// TIA Portal V19 export
FUNCTION "AUTO SUBOUTPUT" : Void   // FC15, LAD
{ S7_Optimized_Access := 'TRUE' }
// stored: SetENOAutomatically false
BEGIN

REGION Network 1: SYRUP MFG VESSEL BOTTOM STERROR RUN
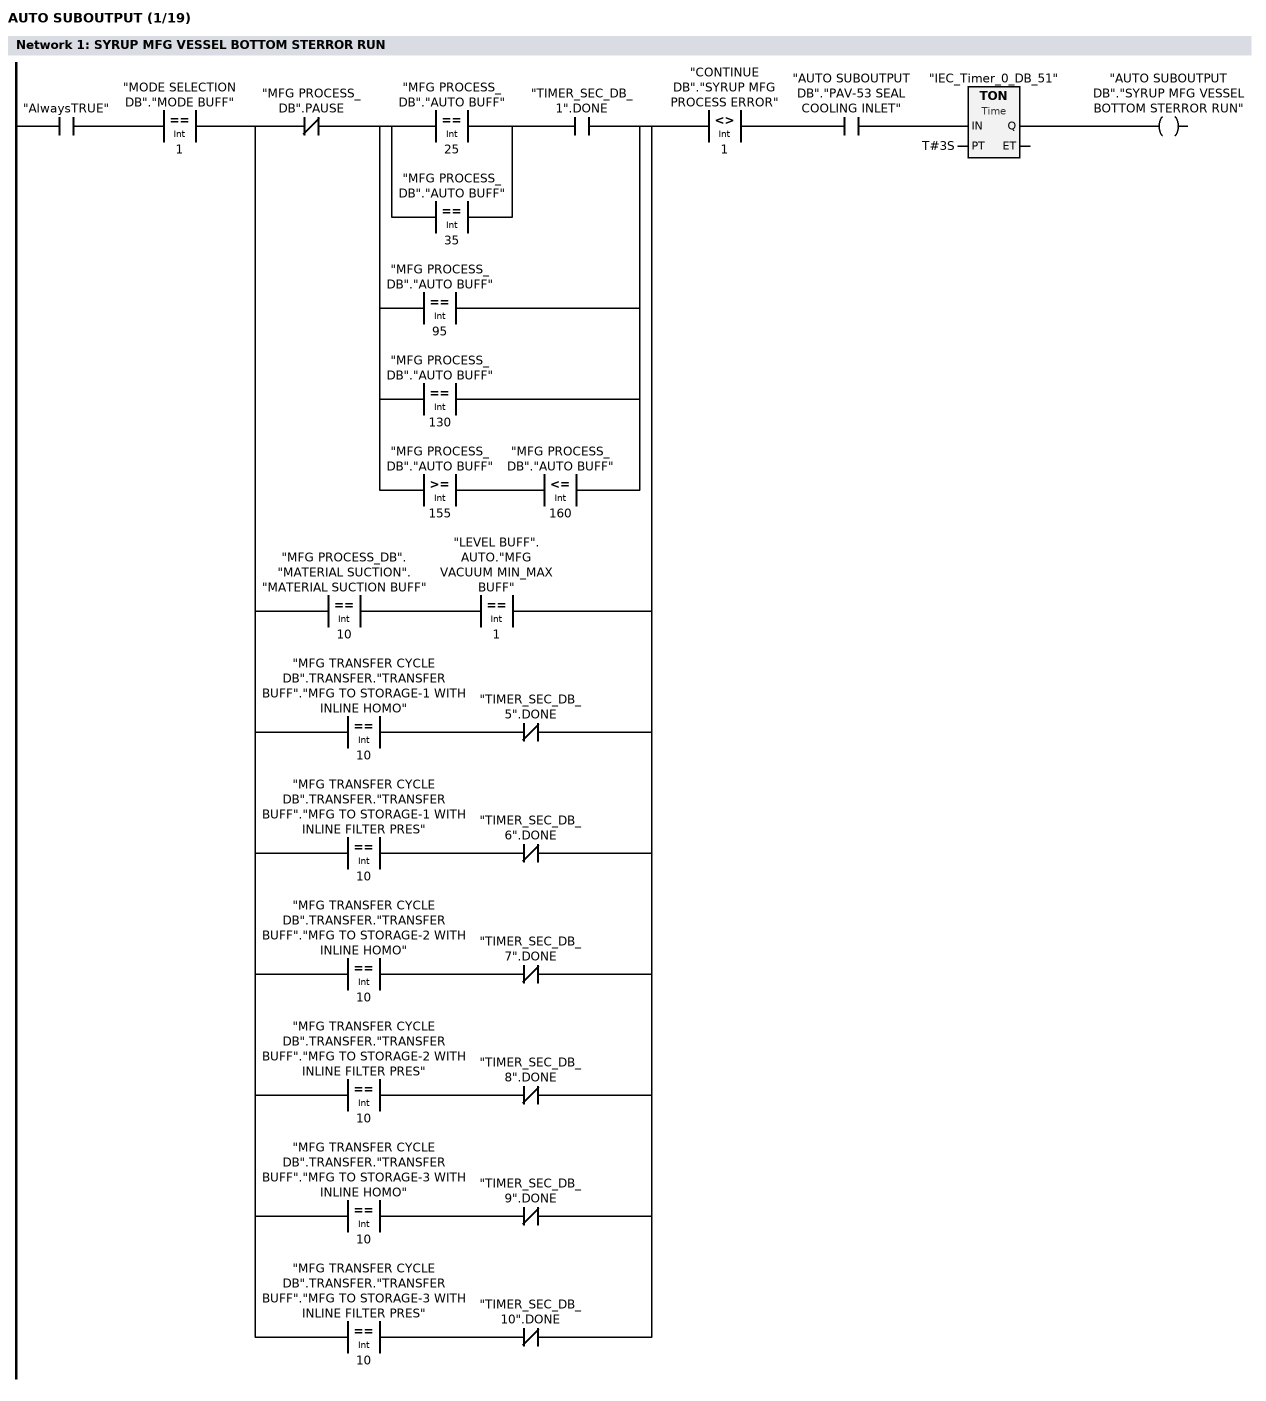
   RUNG wire#powerrail
      Contact( "AlwaysTRUE" )
      { S7_Templates := "SrcType := Int" } EQ_Contact(in1 := "MODE SELECTION DB"."MODE BUFF", in2 := 1)
      wire#w1
      I_Contact( "MFG PROCESS_DB".PAUSE )
      wire#w2
      { S7_Templates := "SrcType := Int" } EQ_Contact(in1 := "MFG PROCESS_DB"."AUTO BUFF", in2 := 25)
      wire#w3
      Contact( "TIMER_SEC_DB_1".DONE )
      wire#w4
      { S7_Templates := "SrcType := Int" } NE_Contact(in1 := "CONTINUE DB"."SYRUP MFG PROCESS ERROR", in2 := 1)
      Contact( "AUTO SUBOUTPUT DB"."PAV-53 SEAL COOLING INLET" )
      { S7_Templates := "time_type := Time" } "IEC_Timer_0_DB_51".TON(pt := T#3S, et =>)
      Coil( "AUTO SUBOUTPUT DB"."SYRUP MFG VESSEL BOTTOM STERROR RUN" )
   END_RUNG
   RUNG wire#w2
      { S7_Templates := "SrcType := Int" } EQ_Contact(in1 := "MFG PROCESS_DB"."AUTO BUFF", in2 := 35)
   END_RUNG wire#w3
   RUNG wire#w2
      { S7_Templates := "SrcType := Int" } EQ_Contact(in1 := "MFG PROCESS_DB"."AUTO BUFF", in2 := 95)
   END_RUNG wire#w4
   RUNG wire#w2
      { S7_Templates := "SrcType := Int" } EQ_Contact(in1 := "MFG PROCESS_DB"."AUTO BUFF", in2 := 130)
   END_RUNG wire#w4
   RUNG wire#w2
      { S7_Templates := "SrcType := Int" } GE_Contact(in1 := "MFG PROCESS_DB"."AUTO BUFF", in2 := 155)
      { S7_Templates := "SrcType := Int" } LE_Contact(in1 := "MFG PROCESS_DB"."AUTO BUFF", in2 := 160)
   END_RUNG wire#w4
   RUNG wire#w1
      { S7_Templates := "SrcType := Int" } EQ_Contact(in1 := "MFG PROCESS_DB"."MATERIAL SUCTION"."MATERIAL SUCTION BUFF", in2 := 10)
      { S7_Templates := "SrcType := Int" } EQ_Contact(in1 := "LEVEL BUFF".AUTO."MFG VACUUM MIN_MAX BUFF", in2 := 1)
   END_RUNG wire#w4
   RUNG wire#w1
      { S7_Templates := "SrcType := Int" } EQ_Contact(in1 := "MFG TRANSFER CYCLE DB".TRANSFER."TRANSFER BUFF"."MFG TO STORAGE-1 WITH INLINE HOMO", in2 := 10)
      I_Contact( "TIMER_SEC_DB_5".DONE )
   END_RUNG wire#w4
   RUNG wire#w1
      { S7_Templates := "SrcType := Int" } EQ_Contact(in1 := "MFG TRANSFER CYCLE DB".TRANSFER."TRANSFER BUFF"."MFG TO STORAGE-1 WITH INLINE FILTER PRES", in2 := 10)
      I_Contact( "TIMER_SEC_DB_6".DONE )
   END_RUNG wire#w4
   RUNG wire#w1
      { S7_Templates := "SrcType := Int" } EQ_Contact(in1 := "MFG TRANSFER CYCLE DB".TRANSFER."TRANSFER BUFF"."MFG TO STORAGE-2 WITH INLINE HOMO", in2 := 10)
      I_Contact( "TIMER_SEC_DB_7".DONE )
   END_RUNG wire#w4
   RUNG wire#w1
      { S7_Templates := "SrcType := Int" } EQ_Contact(in1 := "MFG TRANSFER CYCLE DB".TRANSFER."TRANSFER BUFF"."MFG TO STORAGE-2 WITH INLINE FILTER PRES", in2 := 10)
      I_Contact( "TIMER_SEC_DB_8".DONE )
   END_RUNG wire#w4
   RUNG wire#w1
      { S7_Templates := "SrcType := Int" } EQ_Contact(in1 := "MFG TRANSFER CYCLE DB".TRANSFER."TRANSFER BUFF"."MFG TO STORAGE-3 WITH INLINE HOMO", in2 := 10)
      I_Contact( "TIMER_SEC_DB_9".DONE )
   END_RUNG wire#w4
   RUNG wire#w1
      { S7_Templates := "SrcType := Int" } EQ_Contact(in1 := "MFG TRANSFER CYCLE DB".TRANSFER."TRANSFER BUFF"."MFG TO STORAGE-3 WITH INLINE FILTER PRES", in2 := 10)
      I_Contact( "TIMER_SEC_DB_10".DONE )
   END_RUNG wire#w4
   // the same network as SCL:
   "IEC_Timer_0_DB_51".TON(IN := "AlwaysTRUE" AND ("MODE SELECTION DB"."MODE BUFF" = 1) AND ((NOT "MFG PROCESS_DB".PAUSE AND (((("MFG PROCESS_DB"."AUTO BUFF" = 25) OR ("MFG PROCESS_DB"."AUTO BUFF" = 35)) AND "TIMER_SEC_DB_1".DONE) OR ("MFG PROCESS_DB"."AUTO BUFF" = 95) OR ("MFG PROCESS_DB"."AUTO BUFF" = 130) OR (("MFG PROCESS_DB"."AUTO BUFF" >= 155) AND ("MFG PROCESS_DB"."AUTO BUFF" <= 160)))) OR (("MFG PROCESS_DB"."MATERIAL SUCTION"."MATERIAL SUCTION BUFF" = 10) AND ("LEVEL BUFF".AUTO."MFG VACUUM MIN_MAX BUFF" = 1)) OR (("MFG TRANSFER CYCLE DB".TRANSFER."TRANSFER BUFF"."MFG TO STORAGE-1 WITH INLINE HOMO" = 10) AND NOT "TIMER_SEC_DB_5".DONE) OR (("MFG TRANSFER CYCLE DB".TRANSFER."TRANSFER BUFF"."MFG TO STORAGE-1 WITH INLINE FILTER PRES" = 10) AND NOT "TIMER_SEC_DB_6".DONE) OR (("MFG TRANSFER CYCLE DB".TRANSFER."TRANSFER BUFF"."MFG TO STORAGE-2 WITH INLINE HOMO" = 10) AND NOT "TIMER_SEC_DB_7".DONE) OR (("MFG TRANSFER CYCLE DB".TRANSFER."TRANSFER BUFF"."MFG TO STORAGE-2 WITH INLINE FILTER PRES" = 10) AND NOT "TIMER_SEC_DB_8".DONE) OR (("MFG TRANSFER CYCLE DB".TRANSFER."TRANSFER BUFF"."MFG TO STORAGE-3 WITH INLINE HOMO" = 10) AND NOT "TIMER_SEC_DB_9".DONE) OR (("MFG TRANSFER CYCLE DB".TRANSFER."TRANSFER BUFF"."MFG TO STORAGE-3 WITH INLINE FILTER PRES" = 10) AND NOT "TIMER_SEC_DB_10".DONE)) AND ("CONTINUE DB"."SYRUP MFG PROCESS ERROR" <> 1) AND "AUTO SUBOUTPUT DB"."PAV-53 SEAL COOLING INLET",
                           PT := T#3S);
   "AUTO SUBOUTPUT DB"."SYRUP MFG VESSEL BOTTOM STERROR RUN" := "IEC_Timer_0_DB_51".Q;
END_REGION

REGION Network 2: PREMIXING VESSEL BOTTOM STERROR RUN
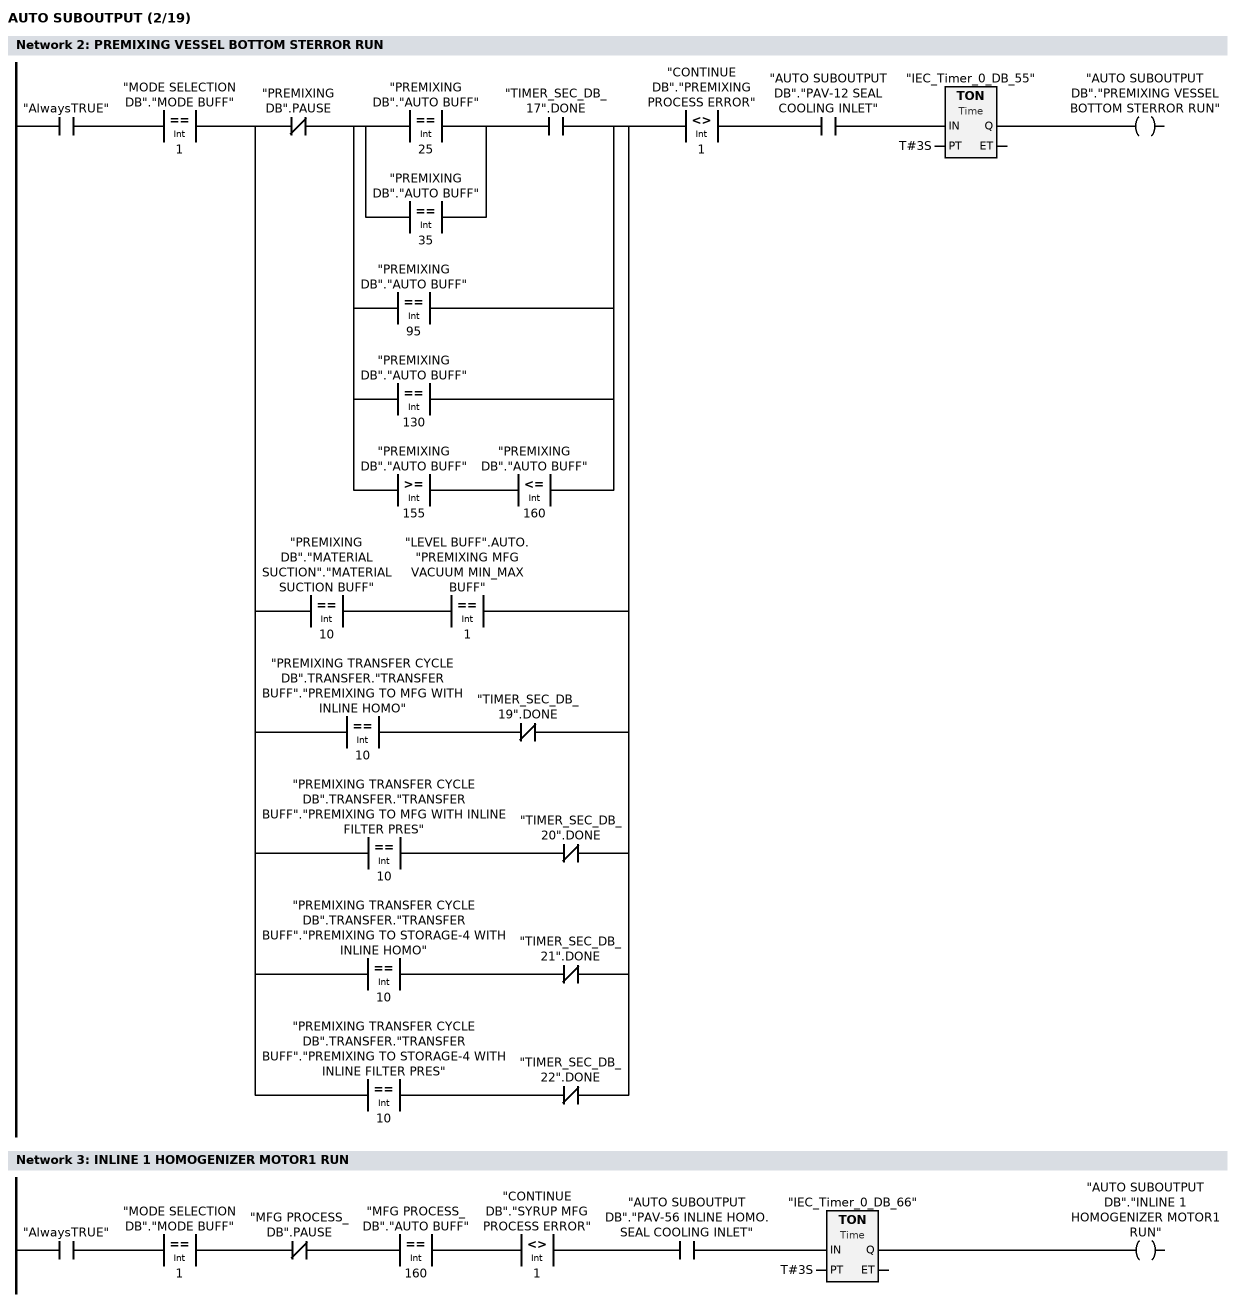
   RUNG wire#powerrail
      Contact( "AlwaysTRUE" )
      { S7_Templates := "SrcType := Int" } EQ_Contact(in1 := "MODE SELECTION DB"."MODE BUFF", in2 := 1)
      wire#w1
      I_Contact( "PREMIXING DB".PAUSE )
      wire#w2
      { S7_Templates := "SrcType := Int" } EQ_Contact(in1 := "PREMIXING DB"."AUTO BUFF", in2 := 25)
      wire#w3
      Contact( "TIMER_SEC_DB_17".DONE )
      wire#w4
      { S7_Templates := "SrcType := Int" } NE_Contact(in1 := "CONTINUE DB"."PREMIXING PROCESS ERROR", in2 := 1)
      Contact( "AUTO SUBOUTPUT DB"."PAV-12 SEAL COOLING INLET" )
      { S7_Templates := "time_type := Time" } "IEC_Timer_0_DB_55".TON(pt := T#3S, et =>)
      Coil( "AUTO SUBOUTPUT DB"."PREMIXING VESSEL BOTTOM STERROR RUN" )
   END_RUNG
   RUNG wire#w2
      { S7_Templates := "SrcType := Int" } EQ_Contact(in1 := "PREMIXING DB"."AUTO BUFF", in2 := 35)
   END_RUNG wire#w3
   RUNG wire#w2
      { S7_Templates := "SrcType := Int" } EQ_Contact(in1 := "PREMIXING DB"."AUTO BUFF", in2 := 95)
   END_RUNG wire#w4
   RUNG wire#w2
      { S7_Templates := "SrcType := Int" } EQ_Contact(in1 := "PREMIXING DB"."AUTO BUFF", in2 := 130)
   END_RUNG wire#w4
   RUNG wire#w2
      { S7_Templates := "SrcType := Int" } GE_Contact(in1 := "PREMIXING DB"."AUTO BUFF", in2 := 155)
      { S7_Templates := "SrcType := Int" } LE_Contact(in1 := "PREMIXING DB"."AUTO BUFF", in2 := 160)
   END_RUNG wire#w4
   RUNG wire#w1
      { S7_Templates := "SrcType := Int" } EQ_Contact(in1 := "PREMIXING DB"."MATERIAL SUCTION"."MATERIAL SUCTION BUFF", in2 := 10)
      { S7_Templates := "SrcType := Int" } EQ_Contact(in1 := "LEVEL BUFF".AUTO."PREMIXING MFG VACUUM MIN_MAX BUFF", in2 := 1)
   END_RUNG wire#w4
   RUNG wire#w1
      { S7_Templates := "SrcType := Int" } EQ_Contact(in1 := "PREMIXING TRANSFER CYCLE DB".TRANSFER."TRANSFER BUFF"."PREMIXING TO MFG WITH INLINE HOMO", in2 := 10)
      I_Contact( "TIMER_SEC_DB_19".DONE )
   END_RUNG wire#w4
   RUNG wire#w1
      { S7_Templates := "SrcType := Int" } EQ_Contact(in1 := "PREMIXING TRANSFER CYCLE DB".TRANSFER."TRANSFER BUFF"."PREMIXING TO MFG WITH INLINE FILTER PRES", in2 := 10)
      I_Contact( "TIMER_SEC_DB_20".DONE )
   END_RUNG wire#w4
   RUNG wire#w1
      { S7_Templates := "SrcType := Int" } EQ_Contact(in1 := "PREMIXING TRANSFER CYCLE DB".TRANSFER."TRANSFER BUFF"."PREMIXING TO STORAGE-4 WITH INLINE HOMO", in2 := 10)
      I_Contact( "TIMER_SEC_DB_21".DONE )
   END_RUNG wire#w4
   RUNG wire#w1
      { S7_Templates := "SrcType := Int" } EQ_Contact(in1 := "PREMIXING TRANSFER CYCLE DB".TRANSFER."TRANSFER BUFF"."PREMIXING TO STORAGE-4 WITH INLINE FILTER PRES", in2 := 10)
      I_Contact( "TIMER_SEC_DB_22".DONE )
   END_RUNG wire#w4
   // the same network as SCL:
   "IEC_Timer_0_DB_55".TON(IN := "AlwaysTRUE" AND ("MODE SELECTION DB"."MODE BUFF" = 1) AND ((NOT "PREMIXING DB".PAUSE AND (((("PREMIXING DB"."AUTO BUFF" = 25) OR ("PREMIXING DB"."AUTO BUFF" = 35)) AND "TIMER_SEC_DB_17".DONE) OR ("PREMIXING DB"."AUTO BUFF" = 95) OR ("PREMIXING DB"."AUTO BUFF" = 130) OR (("PREMIXING DB"."AUTO BUFF" >= 155) AND ("PREMIXING DB"."AUTO BUFF" <= 160)))) OR (("PREMIXING DB"."MATERIAL SUCTION"."MATERIAL SUCTION BUFF" = 10) AND ("LEVEL BUFF".AUTO."PREMIXING MFG VACUUM MIN_MAX BUFF" = 1)) OR (("PREMIXING TRANSFER CYCLE DB".TRANSFER."TRANSFER BUFF"."PREMIXING TO MFG WITH INLINE HOMO" = 10) AND NOT "TIMER_SEC_DB_19".DONE) OR (("PREMIXING TRANSFER CYCLE DB".TRANSFER."TRANSFER BUFF"."PREMIXING TO MFG WITH INLINE FILTER PRES" = 10) AND NOT "TIMER_SEC_DB_20".DONE) OR (("PREMIXING TRANSFER CYCLE DB".TRANSFER."TRANSFER BUFF"."PREMIXING TO STORAGE-4 WITH INLINE HOMO" = 10) AND NOT "TIMER_SEC_DB_21".DONE) OR (("PREMIXING TRANSFER CYCLE DB".TRANSFER."TRANSFER BUFF"."PREMIXING TO STORAGE-4 WITH INLINE FILTER PRES" = 10) AND NOT "TIMER_SEC_DB_22".DONE)) AND ("CONTINUE DB"."PREMIXING PROCESS ERROR" <> 1) AND "AUTO SUBOUTPUT DB"."PAV-12 SEAL COOLING INLET",
                           PT := T#3S);
   "AUTO SUBOUTPUT DB"."PREMIXING VESSEL BOTTOM STERROR RUN" := "IEC_Timer_0_DB_55".Q;
END_REGION

REGION Network 3: INLINE 1 HOMOGENIZER MOTOR1 RUN
   RUNG wire#powerrail
      Contact( "AlwaysTRUE" )
      { S7_Templates := "SrcType := Int" } EQ_Contact(in1 := "MODE SELECTION DB"."MODE BUFF", in2 := 1)
      I_Contact( "MFG PROCESS_DB".PAUSE )
      { S7_Templates := "SrcType := Int" } EQ_Contact(in1 := "MFG PROCESS_DB"."AUTO BUFF", in2 := 160)
      { S7_Templates := "SrcType := Int" } NE_Contact(in1 := "CONTINUE DB"."SYRUP MFG PROCESS ERROR", in2 := 1)
      Contact( "AUTO SUBOUTPUT DB"."PAV-56 INLINE HOMO. SEAL COOLING INLET" )
      { S7_Templates := "time_type := Time" } "IEC_Timer_0_DB_66".TON(pt := T#3S, et =>)
      Coil( "AUTO SUBOUTPUT DB"."INLINE 1 HOMOGENIZER MOTOR1 RUN" )
   END_RUNG
   // the same network as SCL:
   "IEC_Timer_0_DB_66".TON(IN := "AlwaysTRUE" AND ("MODE SELECTION DB"."MODE BUFF" = 1) AND NOT "MFG PROCESS_DB".PAUSE AND ("MFG PROCESS_DB"."AUTO BUFF" = 160) AND ("CONTINUE DB"."SYRUP MFG PROCESS ERROR" <> 1) AND "AUTO SUBOUTPUT DB"."PAV-56 INLINE HOMO. SEAL COOLING INLET",
                           PT := T#3S);
   "AUTO SUBOUTPUT DB"."INLINE 1 HOMOGENIZER MOTOR1 RUN" := "IEC_Timer_0_DB_66".Q;
END_REGION

REGION Network 4: INLINE 2 HOMOGENIZER MOTOR 2 RUN
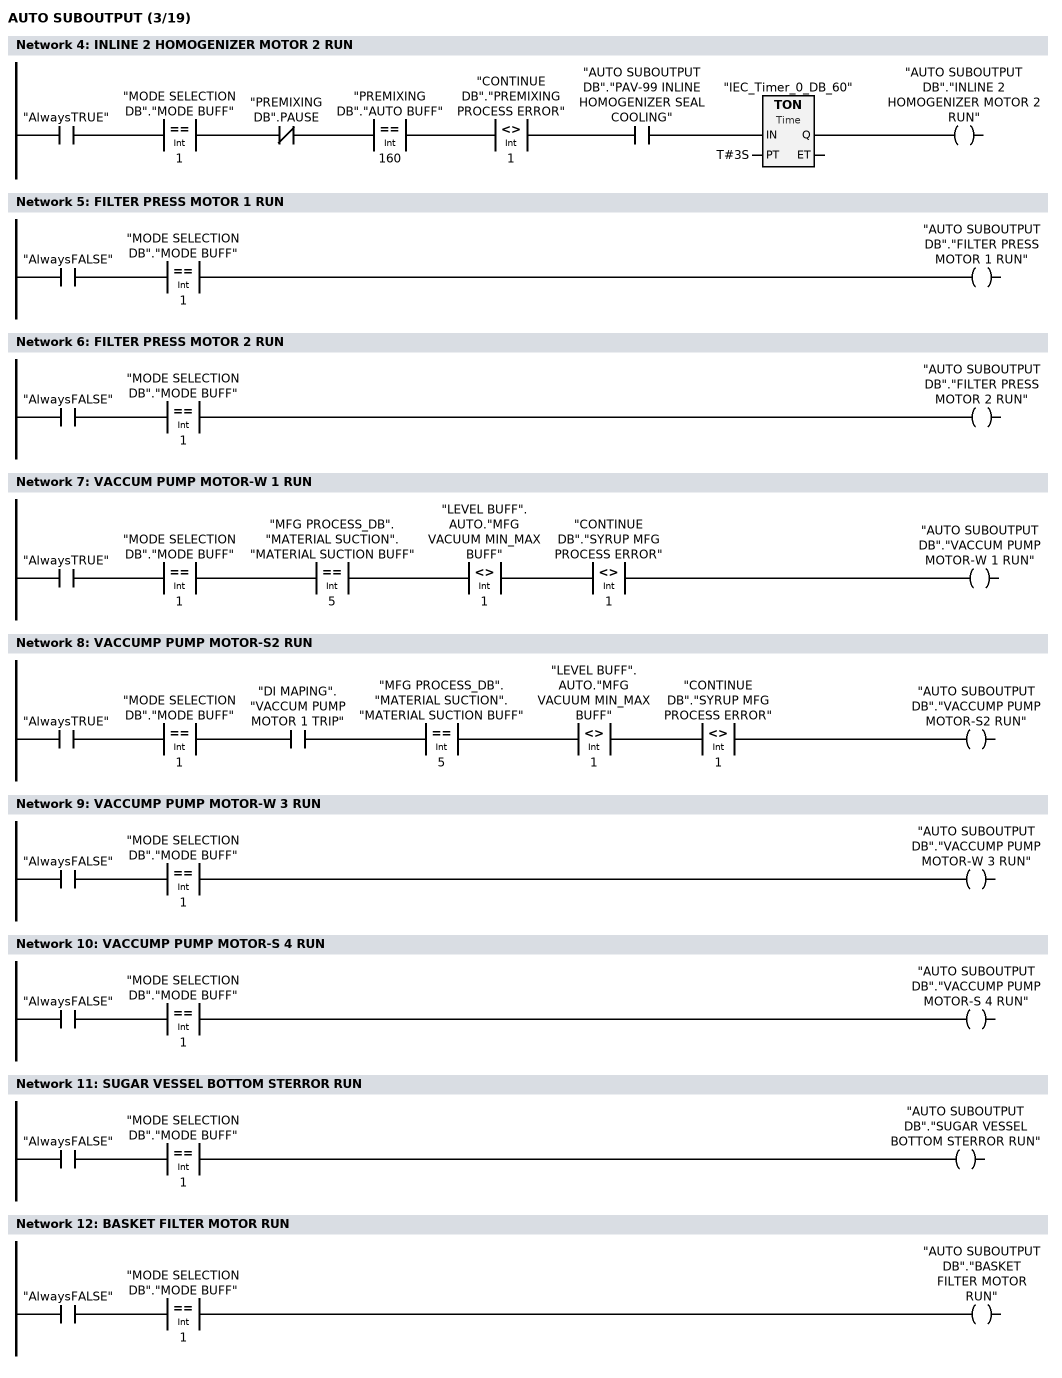
   RUNG wire#powerrail
      Contact( "AlwaysTRUE" )
      { S7_Templates := "SrcType := Int" } EQ_Contact(in1 := "MODE SELECTION DB"."MODE BUFF", in2 := 1)
      I_Contact( "PREMIXING DB".PAUSE )
      { S7_Templates := "SrcType := Int" } EQ_Contact(in1 := "PREMIXING DB"."AUTO BUFF", in2 := 160)
      { S7_Templates := "SrcType := Int" } NE_Contact(in1 := "CONTINUE DB"."PREMIXING PROCESS ERROR", in2 := 1)
      Contact( "AUTO SUBOUTPUT DB"."PAV-99 INLINE HOMOGENIZER SEAL COOLING" )
      { S7_Templates := "time_type := Time" } "IEC_Timer_0_DB_60".TON(pt := T#3S, et =>)
      Coil( "AUTO SUBOUTPUT DB"."INLINE 2 HOMOGENIZER MOTOR 2 RUN" )
   END_RUNG
   // the same network as SCL:
   "IEC_Timer_0_DB_60".TON(IN := "AlwaysTRUE" AND ("MODE SELECTION DB"."MODE BUFF" = 1) AND NOT "PREMIXING DB".PAUSE AND ("PREMIXING DB"."AUTO BUFF" = 160) AND ("CONTINUE DB"."PREMIXING PROCESS ERROR" <> 1) AND "AUTO SUBOUTPUT DB"."PAV-99 INLINE HOMOGENIZER SEAL COOLING",
                           PT := T#3S);
   "AUTO SUBOUTPUT DB"."INLINE 2 HOMOGENIZER MOTOR 2 RUN" := "IEC_Timer_0_DB_60".Q;
END_REGION

REGION Network 5: FILTER PRESS MOTOR 1 RUN
   RUNG wire#powerrail
      Contact( "AlwaysFALSE" )
      { S7_Templates := "SrcType := Int" } EQ_Contact(in1 := "MODE SELECTION DB"."MODE BUFF", in2 := 1)
      Coil( "AUTO SUBOUTPUT DB"."FILTER PRESS MOTOR 1 RUN" )
   END_RUNG
   // the same network as SCL:
   "AUTO SUBOUTPUT DB"."FILTER PRESS MOTOR 1 RUN" := "AlwaysFALSE" AND ("MODE SELECTION DB"."MODE BUFF" = 1);
END_REGION

REGION Network 6: FILTER PRESS MOTOR 2 RUN
   RUNG wire#powerrail
      Contact( "AlwaysFALSE" )
      { S7_Templates := "SrcType := Int" } EQ_Contact(in1 := "MODE SELECTION DB"."MODE BUFF", in2 := 1)
      Coil( "AUTO SUBOUTPUT DB"."FILTER PRESS MOTOR 2 RUN" )
   END_RUNG
   // the same network as SCL:
   "AUTO SUBOUTPUT DB"."FILTER PRESS MOTOR 2 RUN" := "AlwaysFALSE" AND ("MODE SELECTION DB"."MODE BUFF" = 1);
END_REGION

REGION Network 7: VACCUM PUMP MOTOR-W 1 RUN
   RUNG wire#powerrail
      Contact( "AlwaysTRUE" )
      { S7_Templates := "SrcType := Int" } EQ_Contact(in1 := "MODE SELECTION DB"."MODE BUFF", in2 := 1)
      { S7_Templates := "SrcType := Int" } EQ_Contact(in1 := "MFG PROCESS_DB"."MATERIAL SUCTION"."MATERIAL SUCTION BUFF", in2 := 5)
      { S7_Templates := "SrcType := Int" } NE_Contact(in1 := "LEVEL BUFF".AUTO."MFG VACUUM MIN_MAX BUFF", in2 := 1)
      { S7_Templates := "SrcType := Int" } NE_Contact(in1 := "CONTINUE DB"."SYRUP MFG PROCESS ERROR", in2 := 1)
      Coil( "AUTO SUBOUTPUT DB"."VACCUM PUMP MOTOR-W 1 RUN" )
   END_RUNG
   // the same network as SCL:
   "AUTO SUBOUTPUT DB"."VACCUM PUMP MOTOR-W 1 RUN" := "AlwaysTRUE" AND ("MODE SELECTION DB"."MODE BUFF" = 1) AND ("MFG PROCESS_DB"."MATERIAL SUCTION"."MATERIAL SUCTION BUFF" = 5) AND ("LEVEL BUFF".AUTO."MFG VACUUM MIN_MAX BUFF" <> 1) AND ("CONTINUE DB"."SYRUP MFG PROCESS ERROR" <> 1);
END_REGION

REGION Network 8: VACCUMP PUMP MOTOR-S2 RUN
   RUNG wire#powerrail
      Contact( "AlwaysTRUE" )
      { S7_Templates := "SrcType := Int" } EQ_Contact(in1 := "MODE SELECTION DB"."MODE BUFF", in2 := 1)
      Contact( "DI MAPING"."VACCUM PUMP MOTOR 1 TRIP" )
      { S7_Templates := "SrcType := Int" } EQ_Contact(in1 := "MFG PROCESS_DB"."MATERIAL SUCTION"."MATERIAL SUCTION BUFF", in2 := 5)
      { S7_Templates := "SrcType := Int" } NE_Contact(in1 := "LEVEL BUFF".AUTO."MFG VACUUM MIN_MAX BUFF", in2 := 1)
      { S7_Templates := "SrcType := Int" } NE_Contact(in1 := "CONTINUE DB"."SYRUP MFG PROCESS ERROR", in2 := 1)
      Coil( "AUTO SUBOUTPUT DB"."VACCUMP PUMP MOTOR-S2 RUN" )
   END_RUNG
   // the same network as SCL:
   "AUTO SUBOUTPUT DB"."VACCUMP PUMP MOTOR-S2 RUN" := "AlwaysTRUE" AND ("MODE SELECTION DB"."MODE BUFF" = 1) AND "DI MAPING"."VACCUM PUMP MOTOR 1 TRIP" AND ("MFG PROCESS_DB"."MATERIAL SUCTION"."MATERIAL SUCTION BUFF" = 5) AND ("LEVEL BUFF".AUTO."MFG VACUUM MIN_MAX BUFF" <> 1) AND ("CONTINUE DB"."SYRUP MFG PROCESS ERROR" <> 1);
END_REGION

REGION Network 9: VACCUMP PUMP MOTOR-W 3 RUN
   RUNG wire#powerrail
      Contact( "AlwaysFALSE" )
      { S7_Templates := "SrcType := Int" } EQ_Contact(in1 := "MODE SELECTION DB"."MODE BUFF", in2 := 1)
      Coil( "AUTO SUBOUTPUT DB"."VACCUMP PUMP MOTOR-W 3 RUN" )
   END_RUNG
   // the same network as SCL:
   "AUTO SUBOUTPUT DB"."VACCUMP PUMP MOTOR-W 3 RUN" := "AlwaysFALSE" AND ("MODE SELECTION DB"."MODE BUFF" = 1);
END_REGION

REGION Network 10: VACCUMP PUMP MOTOR-S 4 RUN
   RUNG wire#powerrail
      Contact( "AlwaysFALSE" )
      { S7_Templates := "SrcType := Int" } EQ_Contact(in1 := "MODE SELECTION DB"."MODE BUFF", in2 := 1)
      Coil( "AUTO SUBOUTPUT DB"."VACCUMP PUMP MOTOR-S 4 RUN" )
   END_RUNG
   // the same network as SCL:
   "AUTO SUBOUTPUT DB"."VACCUMP PUMP MOTOR-S 4 RUN" := "AlwaysFALSE" AND ("MODE SELECTION DB"."MODE BUFF" = 1);
END_REGION

REGION Network 11: SUGAR VESSEL BOTTOM STERROR RUN
   RUNG wire#powerrail
      Contact( "AlwaysFALSE" )
      { S7_Templates := "SrcType := Int" } EQ_Contact(in1 := "MODE SELECTION DB"."MODE BUFF", in2 := 1)
      Coil( "AUTO SUBOUTPUT DB"."SUGAR VESSEL BOTTOM STERROR RUN" )
   END_RUNG
   // the same network as SCL:
   "AUTO SUBOUTPUT DB"."SUGAR VESSEL BOTTOM STERROR RUN" := "AlwaysFALSE" AND ("MODE SELECTION DB"."MODE BUFF" = 1);
END_REGION

REGION Network 12: BASKET FILTER MOTOR RUN
   RUNG wire#powerrail
      Contact( "AlwaysFALSE" )
      { S7_Templates := "SrcType := Int" } EQ_Contact(in1 := "MODE SELECTION DB"."MODE BUFF", in2 := 1)
      Coil( "AUTO SUBOUTPUT DB"."BASKET FILTER MOTOR RUN" )
   END_RUNG
   // the same network as SCL:
   "AUTO SUBOUTPUT DB"."BASKET FILTER MOTOR RUN" := "AlwaysFALSE" AND ("MODE SELECTION DB"."MODE BUFF" = 1);
END_REGION

REGION Network 13: PBV-01 INGREDIENT INLET
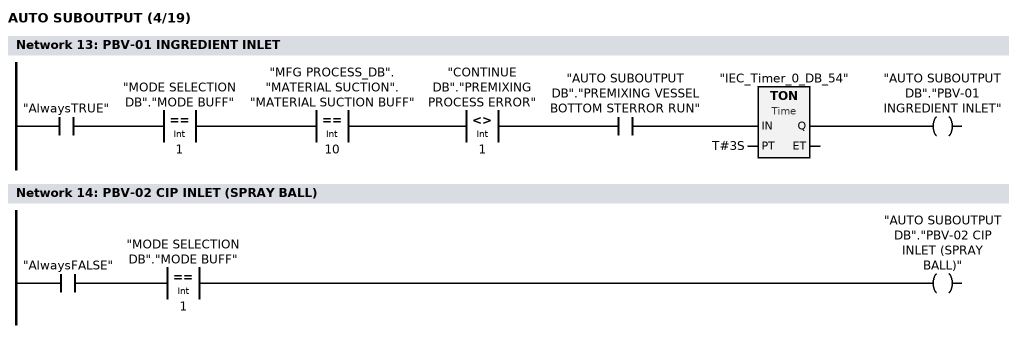
   RUNG wire#powerrail
      Contact( "AlwaysTRUE" )
      { S7_Templates := "SrcType := Int" } EQ_Contact(in1 := "MODE SELECTION DB"."MODE BUFF", in2 := 1)
      { S7_Templates := "SrcType := Int" } EQ_Contact(in1 := "MFG PROCESS_DB"."MATERIAL SUCTION"."MATERIAL SUCTION BUFF", in2 := 10)
      { S7_Templates := "SrcType := Int" } NE_Contact(in1 := "CONTINUE DB"."PREMIXING PROCESS ERROR", in2 := 1)
      Contact( "AUTO SUBOUTPUT DB"."PREMIXING VESSEL BOTTOM STERROR RUN" )
      { S7_Templates := "time_type := Time" } "IEC_Timer_0_DB_54".TON(pt := T#3S, et =>)
      Coil( "AUTO SUBOUTPUT DB"."PBV-01 INGREDIENT INLET" )
   END_RUNG
   // the same network as SCL:
   "IEC_Timer_0_DB_54".TON(IN := "AlwaysTRUE" AND ("MODE SELECTION DB"."MODE BUFF" = 1) AND ("MFG PROCESS_DB"."MATERIAL SUCTION"."MATERIAL SUCTION BUFF" = 10) AND ("CONTINUE DB"."PREMIXING PROCESS ERROR" <> 1) AND "AUTO SUBOUTPUT DB"."PREMIXING VESSEL BOTTOM STERROR RUN",
                           PT := T#3S);
   "AUTO SUBOUTPUT DB"."PBV-01 INGREDIENT INLET" := "IEC_Timer_0_DB_54".Q;
END_REGION

REGION Network 14: PBV-02 CIP INLET (SPRAY BALL)
   RUNG wire#powerrail
      Contact( "AlwaysFALSE" )
      { S7_Templates := "SrcType := Int" } EQ_Contact(in1 := "MODE SELECTION DB"."MODE BUFF", in2 := 1)
      Coil( "AUTO SUBOUTPUT DB"."PBV-02 CIP INLET (SPRAY BALL)" )
   END_RUNG
   // the same network as SCL:
   "AUTO SUBOUTPUT DB"."PBV-02 CIP INLET (SPRAY BALL)" := "AlwaysFALSE" AND ("MODE SELECTION DB"."MODE BUFF" = 1);
END_REGION

REGION Network 15: PBV-03 VENT FILTER ISOLATION
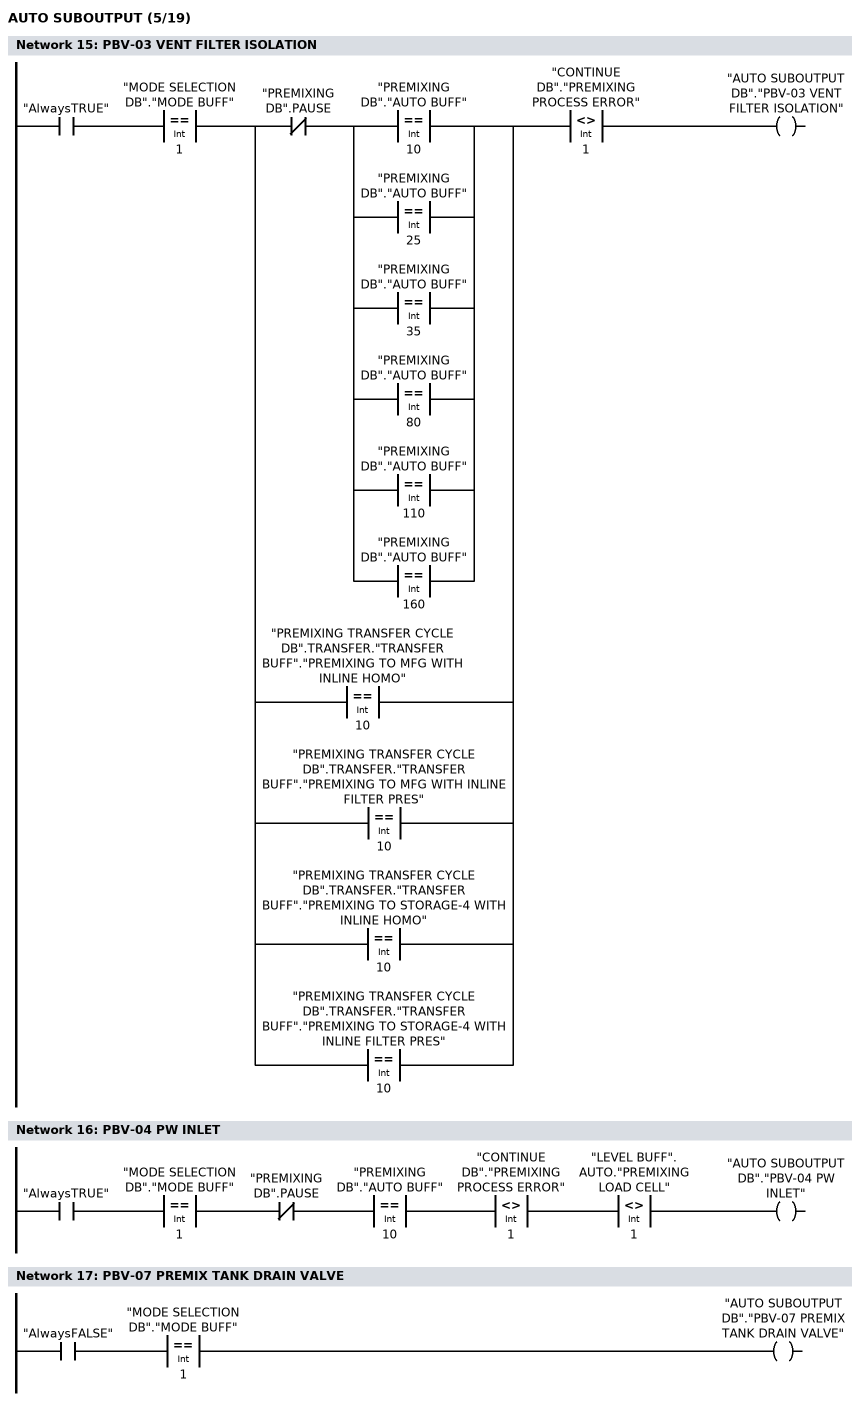
   RUNG wire#powerrail
      Contact( "AlwaysTRUE" )
      { S7_Templates := "SrcType := Int" } EQ_Contact(in1 := "MODE SELECTION DB"."MODE BUFF", in2 := 1)
      wire#w1
      I_Contact( "PREMIXING DB".PAUSE )
      wire#w2
      { S7_Templates := "SrcType := Int" } EQ_Contact(in1 := "PREMIXING DB"."AUTO BUFF", in2 := 10)
      wire#w3
      { S7_Templates := "SrcType := Int" } NE_Contact(in1 := "CONTINUE DB"."PREMIXING PROCESS ERROR", in2 := 1)
      Coil( "AUTO SUBOUTPUT DB"."PBV-03 VENT FILTER ISOLATION" )
   END_RUNG
   RUNG wire#w2
      { S7_Templates := "SrcType := Int" } EQ_Contact(in1 := "PREMIXING DB"."AUTO BUFF", in2 := 25)
   END_RUNG wire#w3
   RUNG wire#w2
      { S7_Templates := "SrcType := Int" } EQ_Contact(in1 := "PREMIXING DB"."AUTO BUFF", in2 := 35)
   END_RUNG wire#w3
   RUNG wire#w2
      { S7_Templates := "SrcType := Int" } EQ_Contact(in1 := "PREMIXING DB"."AUTO BUFF", in2 := 80)
   END_RUNG wire#w3
   RUNG wire#w2
      { S7_Templates := "SrcType := Int" } EQ_Contact(in1 := "PREMIXING DB"."AUTO BUFF", in2 := 110)
   END_RUNG wire#w3
   RUNG wire#w2
      { S7_Templates := "SrcType := Int" } EQ_Contact(in1 := "PREMIXING DB"."AUTO BUFF", in2 := 160)
   END_RUNG wire#w3
   RUNG wire#w1
      { S7_Templates := "SrcType := Int" } EQ_Contact(in1 := "PREMIXING TRANSFER CYCLE DB".TRANSFER."TRANSFER BUFF"."PREMIXING TO MFG WITH INLINE HOMO", in2 := 10)
   END_RUNG wire#w3
   RUNG wire#w1
      { S7_Templates := "SrcType := Int" } EQ_Contact(in1 := "PREMIXING TRANSFER CYCLE DB".TRANSFER."TRANSFER BUFF"."PREMIXING TO MFG WITH INLINE FILTER PRES", in2 := 10)
   END_RUNG wire#w3
   RUNG wire#w1
      { S7_Templates := "SrcType := Int" } EQ_Contact(in1 := "PREMIXING TRANSFER CYCLE DB".TRANSFER."TRANSFER BUFF"."PREMIXING TO STORAGE-4 WITH INLINE HOMO", in2 := 10)
   END_RUNG wire#w3
   RUNG wire#w1
      { S7_Templates := "SrcType := Int" } EQ_Contact(in1 := "PREMIXING TRANSFER CYCLE DB".TRANSFER."TRANSFER BUFF"."PREMIXING TO STORAGE-4 WITH INLINE FILTER PRES", in2 := 10)
   END_RUNG wire#w3
   // the same network as SCL:
   "AUTO SUBOUTPUT DB"."PBV-03 VENT FILTER ISOLATION" := "AlwaysTRUE" AND ("MODE SELECTION DB"."MODE BUFF" = 1) AND ((NOT "PREMIXING DB".PAUSE AND (("PREMIXING DB"."AUTO BUFF" = 10) OR ("PREMIXING DB"."AUTO BUFF" = 25) OR ("PREMIXING DB"."AUTO BUFF" = 35) OR ("PREMIXING DB"."AUTO BUFF" = 80) OR ("PREMIXING DB"."AUTO BUFF" = 110) OR ("PREMIXING DB"."AUTO BUFF" = 160))) OR ("PREMIXING TRANSFER CYCLE DB".TRANSFER."TRANSFER BUFF"."PREMIXING TO MFG WITH INLINE HOMO" = 10) OR ("PREMIXING TRANSFER CYCLE DB".TRANSFER."TRANSFER BUFF"."PREMIXING TO MFG WITH INLINE FILTER PRES" = 10) OR ("PREMIXING TRANSFER CYCLE DB".TRANSFER."TRANSFER BUFF"."PREMIXING TO STORAGE-4 WITH INLINE HOMO" = 10) OR ("PREMIXING TRANSFER CYCLE DB".TRANSFER."TRANSFER BUFF"."PREMIXING TO STORAGE-4 WITH INLINE FILTER PRES" = 10)) AND ("CONTINUE DB"."PREMIXING PROCESS ERROR" <> 1);
END_REGION

REGION Network 16: PBV-04 PW INLET
   RUNG wire#powerrail
      Contact( "AlwaysTRUE" )
      { S7_Templates := "SrcType := Int" } EQ_Contact(in1 := "MODE SELECTION DB"."MODE BUFF", in2 := 1)
      I_Contact( "PREMIXING DB".PAUSE )
      { S7_Templates := "SrcType := Int" } EQ_Contact(in1 := "PREMIXING DB"."AUTO BUFF", in2 := 10)
      { S7_Templates := "SrcType := Int" } NE_Contact(in1 := "CONTINUE DB"."PREMIXING PROCESS ERROR", in2 := 1)
      { S7_Templates := "SrcType := Int" } NE_Contact(in1 := "LEVEL BUFF".AUTO."PREMIXING LOAD CELL", in2 := 1)
      Coil( "AUTO SUBOUTPUT DB"."PBV-04 PW INLET" )
   END_RUNG
   // the same network as SCL:
   "AUTO SUBOUTPUT DB"."PBV-04 PW INLET" := "AlwaysTRUE" AND ("MODE SELECTION DB"."MODE BUFF" = 1) AND NOT "PREMIXING DB".PAUSE AND ("PREMIXING DB"."AUTO BUFF" = 10) AND ("CONTINUE DB"."PREMIXING PROCESS ERROR" <> 1) AND ("LEVEL BUFF".AUTO."PREMIXING LOAD CELL" <> 1);
END_REGION

REGION Network 17: PBV-07 PREMIX TANK DRAIN VALVE
   RUNG wire#powerrail
      Contact( "AlwaysFALSE" )
      { S7_Templates := "SrcType := Int" } EQ_Contact(in1 := "MODE SELECTION DB"."MODE BUFF", in2 := 1)
      Coil( "AUTO SUBOUTPUT DB"."PBV-07 PREMIX TANK DRAIN VALVE" )
   END_RUNG
   // the same network as SCL:
   "AUTO SUBOUTPUT DB"."PBV-07 PREMIX TANK DRAIN VALVE" := "AlwaysFALSE" AND ("MODE SELECTION DB"."MODE BUFF" = 1);
END_REGION

REGION Network 18: PAV-09 JACKET STEAM INLET
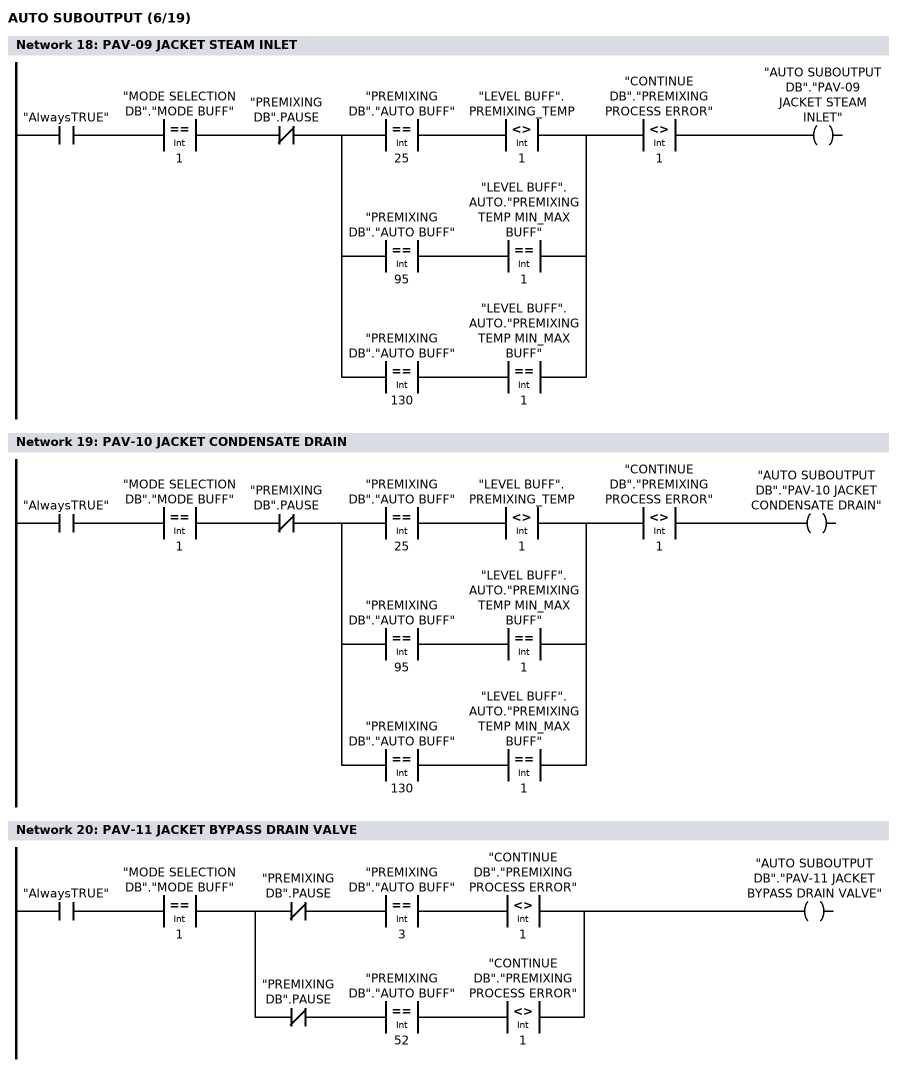
   RUNG wire#powerrail
      Contact( "AlwaysTRUE" )
      { S7_Templates := "SrcType := Int" } EQ_Contact(in1 := "MODE SELECTION DB"."MODE BUFF", in2 := 1)
      I_Contact( "PREMIXING DB".PAUSE )
      wire#w1
      { S7_Templates := "SrcType := Int" } EQ_Contact(in1 := "PREMIXING DB"."AUTO BUFF", in2 := 25)
      { S7_Templates := "SrcType := Int" } NE_Contact(in1 := "LEVEL BUFF".PREMIXING_TEMP, in2 := 1)
      wire#w2
      { S7_Templates := "SrcType := Int" } NE_Contact(in1 := "CONTINUE DB"."PREMIXING PROCESS ERROR", in2 := 1)
      Coil( "AUTO SUBOUTPUT DB"."PAV-09 JACKET STEAM INLET" )
   END_RUNG
   RUNG wire#w1
      { S7_Templates := "SrcType := Int" } EQ_Contact(in1 := "PREMIXING DB"."AUTO BUFF", in2 := 95)
      { S7_Templates := "SrcType := Int" } EQ_Contact(in1 := "LEVEL BUFF".AUTO."PREMIXING TEMP MIN_MAX BUFF", in2 := 1)
   END_RUNG wire#w2
   RUNG wire#w1
      { S7_Templates := "SrcType := Int" } EQ_Contact(in1 := "PREMIXING DB"."AUTO BUFF", in2 := 130)
      { S7_Templates := "SrcType := Int" } EQ_Contact(in1 := "LEVEL BUFF".AUTO."PREMIXING TEMP MIN_MAX BUFF", in2 := 1)
   END_RUNG wire#w2
   // the same network as SCL:
   "AUTO SUBOUTPUT DB"."PAV-09 JACKET STEAM INLET" := "AlwaysTRUE" AND ("MODE SELECTION DB"."MODE BUFF" = 1) AND NOT "PREMIXING DB".PAUSE AND ((("PREMIXING DB"."AUTO BUFF" = 25) AND ("LEVEL BUFF".PREMIXING_TEMP <> 1)) OR (("PREMIXING DB"."AUTO BUFF" = 95) AND ("LEVEL BUFF".AUTO."PREMIXING TEMP MIN_MAX BUFF" = 1)) OR (("PREMIXING DB"."AUTO BUFF" = 130) AND ("LEVEL BUFF".AUTO."PREMIXING TEMP MIN_MAX BUFF" = 1))) AND ("CONTINUE DB"."PREMIXING PROCESS ERROR" <> 1);
END_REGION

REGION Network 19: PAV-10 JACKET CONDENSATE DRAIN
   RUNG wire#powerrail
      Contact( "AlwaysTRUE" )
      { S7_Templates := "SrcType := Int" } EQ_Contact(in1 := "MODE SELECTION DB"."MODE BUFF", in2 := 1)
      I_Contact( "PREMIXING DB".PAUSE )
      wire#w1
      { S7_Templates := "SrcType := Int" } EQ_Contact(in1 := "PREMIXING DB"."AUTO BUFF", in2 := 25)
      { S7_Templates := "SrcType := Int" } NE_Contact(in1 := "LEVEL BUFF".PREMIXING_TEMP, in2 := 1)
      wire#w2
      { S7_Templates := "SrcType := Int" } NE_Contact(in1 := "CONTINUE DB"."PREMIXING PROCESS ERROR", in2 := 1)
      Coil( "AUTO SUBOUTPUT DB"."PAV-10 JACKET CONDENSATE DRAIN" )
   END_RUNG
   RUNG wire#w1
      { S7_Templates := "SrcType := Int" } EQ_Contact(in1 := "PREMIXING DB"."AUTO BUFF", in2 := 95)
      { S7_Templates := "SrcType := Int" } EQ_Contact(in1 := "LEVEL BUFF".AUTO."PREMIXING TEMP MIN_MAX BUFF", in2 := 1)
   END_RUNG wire#w2
   RUNG wire#w1
      { S7_Templates := "SrcType := Int" } EQ_Contact(in1 := "PREMIXING DB"."AUTO BUFF", in2 := 130)
      { S7_Templates := "SrcType := Int" } EQ_Contact(in1 := "LEVEL BUFF".AUTO."PREMIXING TEMP MIN_MAX BUFF", in2 := 1)
   END_RUNG wire#w2
   // the same network as SCL:
   "AUTO SUBOUTPUT DB"."PAV-10 JACKET CONDENSATE DRAIN" := "AlwaysTRUE" AND ("MODE SELECTION DB"."MODE BUFF" = 1) AND NOT "PREMIXING DB".PAUSE AND ((("PREMIXING DB"."AUTO BUFF" = 25) AND ("LEVEL BUFF".PREMIXING_TEMP <> 1)) OR (("PREMIXING DB"."AUTO BUFF" = 95) AND ("LEVEL BUFF".AUTO."PREMIXING TEMP MIN_MAX BUFF" = 1)) OR (("PREMIXING DB"."AUTO BUFF" = 130) AND ("LEVEL BUFF".AUTO."PREMIXING TEMP MIN_MAX BUFF" = 1))) AND ("CONTINUE DB"."PREMIXING PROCESS ERROR" <> 1);
END_REGION

REGION Network 20: PAV-11 JACKET BYPASS DRAIN VALVE
   RUNG wire#powerrail
      Contact( "AlwaysTRUE" )
      { S7_Templates := "SrcType := Int" } EQ_Contact(in1 := "MODE SELECTION DB"."MODE BUFF", in2 := 1)
      wire#w1
      I_Contact( "PREMIXING DB".PAUSE )
      { S7_Templates := "SrcType := Int" } EQ_Contact(in1 := "PREMIXING DB"."AUTO BUFF", in2 := 3)
      { S7_Templates := "SrcType := Int" } NE_Contact(in1 := "CONTINUE DB"."PREMIXING PROCESS ERROR", in2 := 1)
      wire#w2
      Coil( "AUTO SUBOUTPUT DB"."PAV-11 JACKET BYPASS DRAIN VALVE" )
   END_RUNG
   RUNG wire#w1
      I_Contact( "PREMIXING DB".PAUSE )
      { S7_Templates := "SrcType := Int" } EQ_Contact(in1 := "PREMIXING DB"."AUTO BUFF", in2 := 52)
      { S7_Templates := "SrcType := Int" } NE_Contact(in1 := "CONTINUE DB"."PREMIXING PROCESS ERROR", in2 := 1)
   END_RUNG wire#w2
   // the same network as SCL:
   "AUTO SUBOUTPUT DB"."PAV-11 JACKET BYPASS DRAIN VALVE" := "AlwaysTRUE" AND ("MODE SELECTION DB"."MODE BUFF" = 1) AND ((NOT "PREMIXING DB".PAUSE AND ("PREMIXING DB"."AUTO BUFF" = 3) AND ("CONTINUE DB"."PREMIXING PROCESS ERROR" <> 1)) OR (NOT "PREMIXING DB".PAUSE AND ("PREMIXING DB"."AUTO BUFF" = 52) AND ("CONTINUE DB"."PREMIXING PROCESS ERROR" <> 1)));
END_REGION

REGION Network 21: PAV-12 SEAL COOLING INLET
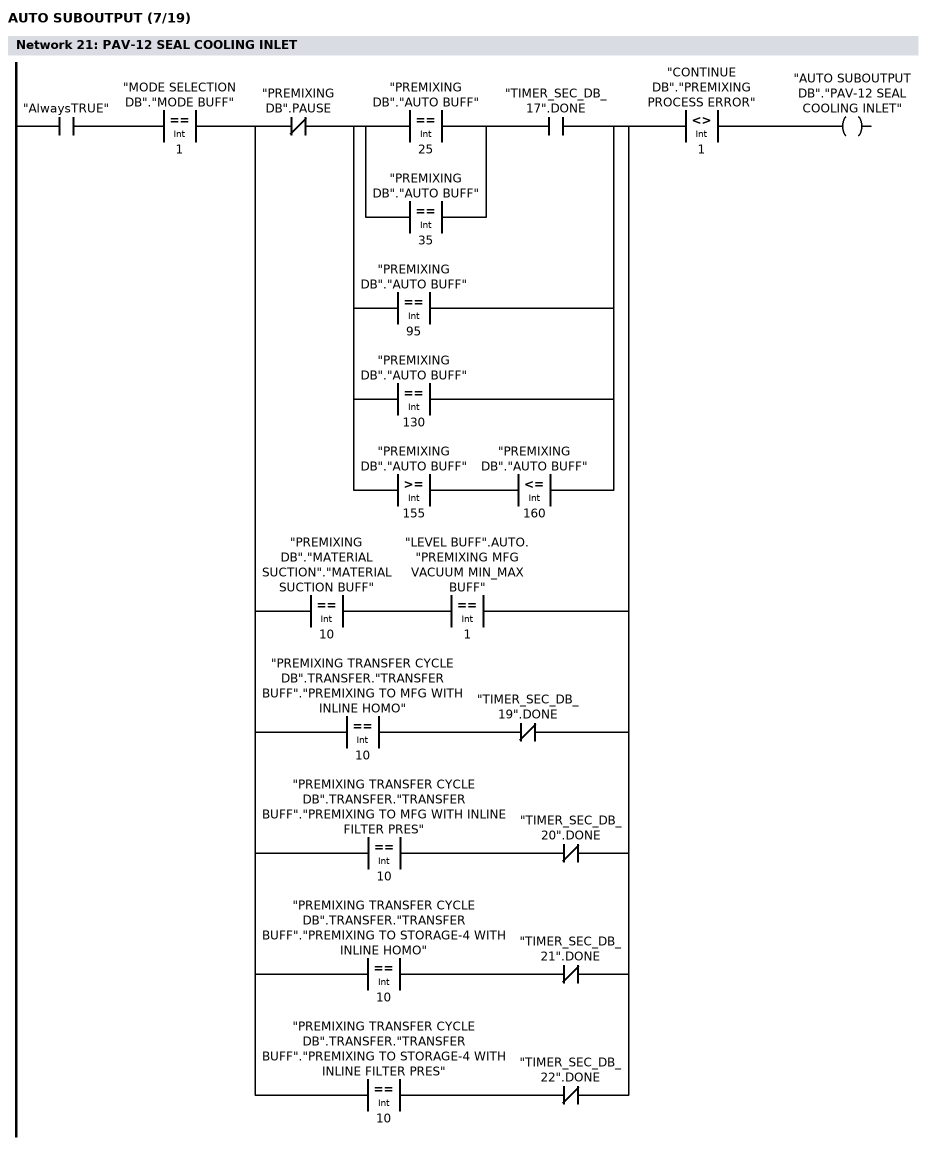
   RUNG wire#powerrail
      Contact( "AlwaysTRUE" )
      { S7_Templates := "SrcType := Int" } EQ_Contact(in1 := "MODE SELECTION DB"."MODE BUFF", in2 := 1)
      wire#w1
      I_Contact( "PREMIXING DB".PAUSE )
      wire#w2
      { S7_Templates := "SrcType := Int" } EQ_Contact(in1 := "PREMIXING DB"."AUTO BUFF", in2 := 25)
      wire#w3
      Contact( "TIMER_SEC_DB_17".DONE )
      wire#w4
      { S7_Templates := "SrcType := Int" } NE_Contact(in1 := "CONTINUE DB"."PREMIXING PROCESS ERROR", in2 := 1)
      Coil( "AUTO SUBOUTPUT DB"."PAV-12 SEAL COOLING INLET" )
   END_RUNG
   RUNG wire#w2
      { S7_Templates := "SrcType := Int" } EQ_Contact(in1 := "PREMIXING DB"."AUTO BUFF", in2 := 35)
   END_RUNG wire#w3
   RUNG wire#w2
      { S7_Templates := "SrcType := Int" } EQ_Contact(in1 := "PREMIXING DB"."AUTO BUFF", in2 := 95)
   END_RUNG wire#w4
   RUNG wire#w2
      { S7_Templates := "SrcType := Int" } EQ_Contact(in1 := "PREMIXING DB"."AUTO BUFF", in2 := 130)
   END_RUNG wire#w4
   RUNG wire#w2
      { S7_Templates := "SrcType := Int" } GE_Contact(in1 := "PREMIXING DB"."AUTO BUFF", in2 := 155)
      { S7_Templates := "SrcType := Int" } LE_Contact(in1 := "PREMIXING DB"."AUTO BUFF", in2 := 160)
   END_RUNG wire#w4
   RUNG wire#w1
      { S7_Templates := "SrcType := Int" } EQ_Contact(in1 := "PREMIXING DB"."MATERIAL SUCTION"."MATERIAL SUCTION BUFF", in2 := 10)
      { S7_Templates := "SrcType := Int" } EQ_Contact(in1 := "LEVEL BUFF".AUTO."PREMIXING MFG VACUUM MIN_MAX BUFF", in2 := 1)
   END_RUNG wire#w4
   RUNG wire#w1
      { S7_Templates := "SrcType := Int" } EQ_Contact(in1 := "PREMIXING TRANSFER CYCLE DB".TRANSFER."TRANSFER BUFF"."PREMIXING TO MFG WITH INLINE HOMO", in2 := 10)
      I_Contact( "TIMER_SEC_DB_19".DONE )
   END_RUNG wire#w4
   RUNG wire#w1
      { S7_Templates := "SrcType := Int" } EQ_Contact(in1 := "PREMIXING TRANSFER CYCLE DB".TRANSFER."TRANSFER BUFF"."PREMIXING TO MFG WITH INLINE FILTER PRES", in2 := 10)
      I_Contact( "TIMER_SEC_DB_20".DONE )
   END_RUNG wire#w4
   RUNG wire#w1
      { S7_Templates := "SrcType := Int" } EQ_Contact(in1 := "PREMIXING TRANSFER CYCLE DB".TRANSFER."TRANSFER BUFF"."PREMIXING TO STORAGE-4 WITH INLINE HOMO", in2 := 10)
      I_Contact( "TIMER_SEC_DB_21".DONE )
   END_RUNG wire#w4
   RUNG wire#w1
      { S7_Templates := "SrcType := Int" } EQ_Contact(in1 := "PREMIXING TRANSFER CYCLE DB".TRANSFER."TRANSFER BUFF"."PREMIXING TO STORAGE-4 WITH INLINE FILTER PRES", in2 := 10)
      I_Contact( "TIMER_SEC_DB_22".DONE )
   END_RUNG wire#w4
   // the same network as SCL:
   "AUTO SUBOUTPUT DB"."PAV-12 SEAL COOLING INLET" := "AlwaysTRUE" AND ("MODE SELECTION DB"."MODE BUFF" = 1) AND ((NOT "PREMIXING DB".PAUSE AND (((("PREMIXING DB"."AUTO BUFF" = 25) OR ("PREMIXING DB"."AUTO BUFF" = 35)) AND "TIMER_SEC_DB_17".DONE) OR ("PREMIXING DB"."AUTO BUFF" = 95) OR ("PREMIXING DB"."AUTO BUFF" = 130) OR (("PREMIXING DB"."AUTO BUFF" >= 155) AND ("PREMIXING DB"."AUTO BUFF" <= 160)))) OR (("PREMIXING DB"."MATERIAL SUCTION"."MATERIAL SUCTION BUFF" = 10) AND ("LEVEL BUFF".AUTO."PREMIXING MFG VACUUM MIN_MAX BUFF" = 1)) OR (("PREMIXING TRANSFER CYCLE DB".TRANSFER."TRANSFER BUFF"."PREMIXING TO MFG WITH INLINE HOMO" = 10) AND NOT "TIMER_SEC_DB_19".DONE) OR (("PREMIXING TRANSFER CYCLE DB".TRANSFER."TRANSFER BUFF"."PREMIXING TO MFG WITH INLINE FILTER PRES" = 10) AND NOT "TIMER_SEC_DB_20".DONE) OR (("PREMIXING TRANSFER CYCLE DB".TRANSFER."TRANSFER BUFF"."PREMIXING TO STORAGE-4 WITH INLINE HOMO" = 10) AND NOT "TIMER_SEC_DB_21".DONE) OR (("PREMIXING TRANSFER CYCLE DB".TRANSFER."TRANSFER BUFF"."PREMIXING TO STORAGE-4 WITH INLINE FILTER PRES" = 10) AND NOT "TIMER_SEC_DB_22".DONE)) AND ("CONTINUE DB"."PREMIXING PROCESS ERROR" <> 1);
END_REGION

REGION Network 22: PAV-13 WATER COOLING INLET
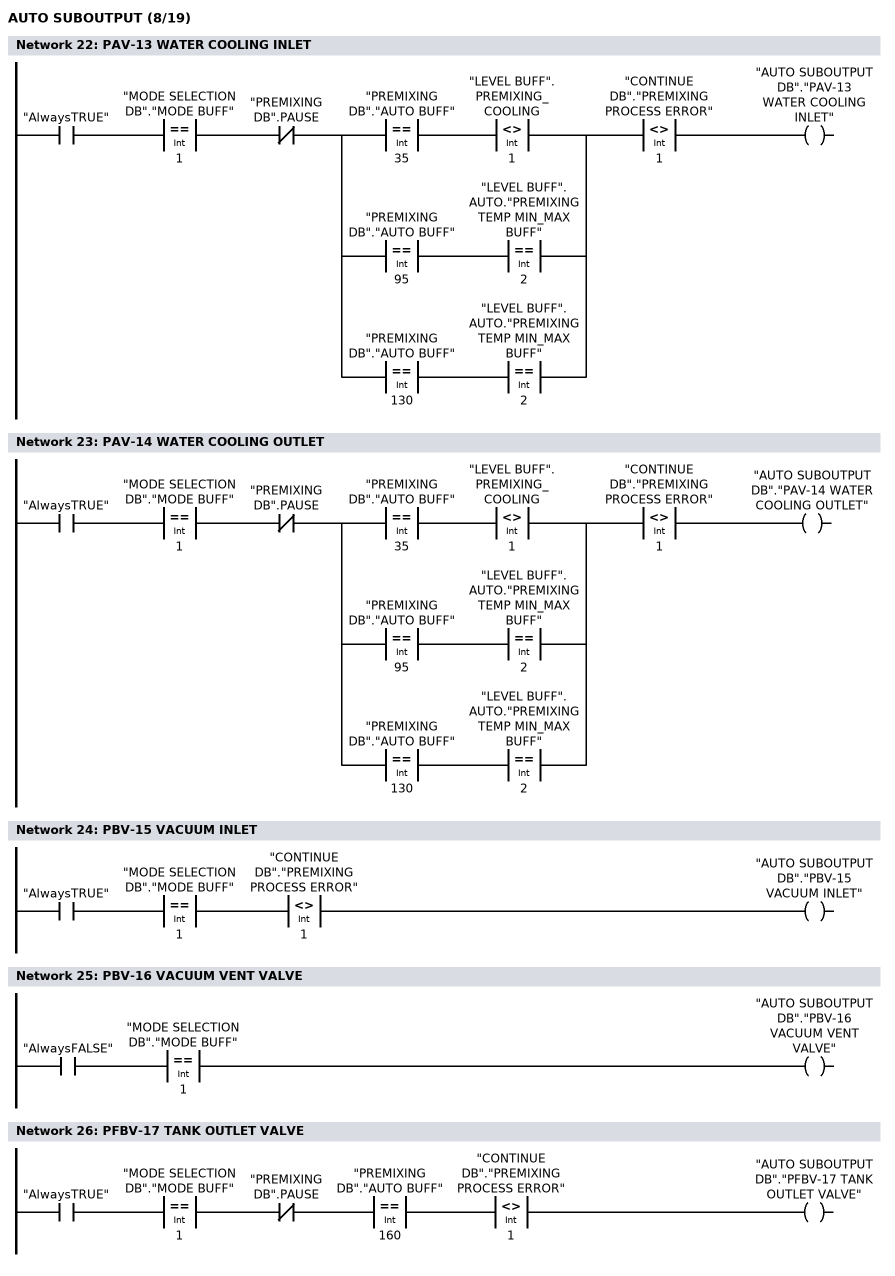
   RUNG wire#powerrail
      Contact( "AlwaysTRUE" )
      { S7_Templates := "SrcType := Int" } EQ_Contact(in1 := "MODE SELECTION DB"."MODE BUFF", in2 := 1)
      I_Contact( "PREMIXING DB".PAUSE )
      wire#w1
      { S7_Templates := "SrcType := Int" } EQ_Contact(in1 := "PREMIXING DB"."AUTO BUFF", in2 := 35)
      { S7_Templates := "SrcType := Int" } NE_Contact(in1 := "LEVEL BUFF".PREMIXING_COOLING, in2 := 1)
      wire#w2
      { S7_Templates := "SrcType := Int" } NE_Contact(in1 := "CONTINUE DB"."PREMIXING PROCESS ERROR", in2 := 1)
      Coil( "AUTO SUBOUTPUT DB"."PAV-13 WATER COOLING INLET" )
   END_RUNG
   RUNG wire#w1
      { S7_Templates := "SrcType := Int" } EQ_Contact(in1 := "PREMIXING DB"."AUTO BUFF", in2 := 95)
      { S7_Templates := "SrcType := Int" } EQ_Contact(in1 := "LEVEL BUFF".AUTO."PREMIXING TEMP MIN_MAX BUFF", in2 := 2)
   END_RUNG wire#w2
   RUNG wire#w1
      { S7_Templates := "SrcType := Int" } EQ_Contact(in1 := "PREMIXING DB"."AUTO BUFF", in2 := 130)
      { S7_Templates := "SrcType := Int" } EQ_Contact(in1 := "LEVEL BUFF".AUTO."PREMIXING TEMP MIN_MAX BUFF", in2 := 2)
   END_RUNG wire#w2
   // the same network as SCL:
   "AUTO SUBOUTPUT DB"."PAV-13 WATER COOLING INLET" := "AlwaysTRUE" AND ("MODE SELECTION DB"."MODE BUFF" = 1) AND NOT "PREMIXING DB".PAUSE AND ((("PREMIXING DB"."AUTO BUFF" = 35) AND ("LEVEL BUFF".PREMIXING_COOLING <> 1)) OR (("PREMIXING DB"."AUTO BUFF" = 95) AND ("LEVEL BUFF".AUTO."PREMIXING TEMP MIN_MAX BUFF" = 2)) OR (("PREMIXING DB"."AUTO BUFF" = 130) AND ("LEVEL BUFF".AUTO."PREMIXING TEMP MIN_MAX BUFF" = 2))) AND ("CONTINUE DB"."PREMIXING PROCESS ERROR" <> 1);
END_REGION

REGION Network 23: PAV-14 WATER COOLING OUTLET
   RUNG wire#powerrail
      Contact( "AlwaysTRUE" )
      { S7_Templates := "SrcType := Int" } EQ_Contact(in1 := "MODE SELECTION DB"."MODE BUFF", in2 := 1)
      I_Contact( "PREMIXING DB".PAUSE )
      wire#w1
      { S7_Templates := "SrcType := Int" } EQ_Contact(in1 := "PREMIXING DB"."AUTO BUFF", in2 := 35)
      { S7_Templates := "SrcType := Int" } NE_Contact(in1 := "LEVEL BUFF".PREMIXING_COOLING, in2 := 1)
      wire#w2
      { S7_Templates := "SrcType := Int" } NE_Contact(in1 := "CONTINUE DB"."PREMIXING PROCESS ERROR", in2 := 1)
      Coil( "AUTO SUBOUTPUT DB"."PAV-14 WATER COOLING OUTLET" )
   END_RUNG
   RUNG wire#w1
      { S7_Templates := "SrcType := Int" } EQ_Contact(in1 := "PREMIXING DB"."AUTO BUFF", in2 := 95)
      { S7_Templates := "SrcType := Int" } EQ_Contact(in1 := "LEVEL BUFF".AUTO."PREMIXING TEMP MIN_MAX BUFF", in2 := 2)
   END_RUNG wire#w2
   RUNG wire#w1
      { S7_Templates := "SrcType := Int" } EQ_Contact(in1 := "PREMIXING DB"."AUTO BUFF", in2 := 130)
      { S7_Templates := "SrcType := Int" } EQ_Contact(in1 := "LEVEL BUFF".AUTO."PREMIXING TEMP MIN_MAX BUFF", in2 := 2)
   END_RUNG wire#w2
   // the same network as SCL:
   "AUTO SUBOUTPUT DB"."PAV-14 WATER COOLING OUTLET" := "AlwaysTRUE" AND ("MODE SELECTION DB"."MODE BUFF" = 1) AND NOT "PREMIXING DB".PAUSE AND ((("PREMIXING DB"."AUTO BUFF" = 35) AND ("LEVEL BUFF".PREMIXING_COOLING <> 1)) OR (("PREMIXING DB"."AUTO BUFF" = 95) AND ("LEVEL BUFF".AUTO."PREMIXING TEMP MIN_MAX BUFF" = 2)) OR (("PREMIXING DB"."AUTO BUFF" = 130) AND ("LEVEL BUFF".AUTO."PREMIXING TEMP MIN_MAX BUFF" = 2))) AND ("CONTINUE DB"."PREMIXING PROCESS ERROR" <> 1);
END_REGION

REGION Network 24: PBV-15 VACUUM INLET
   RUNG wire#powerrail
      Contact( "AlwaysTRUE" )
      { S7_Templates := "SrcType := Int" } EQ_Contact(in1 := "MODE SELECTION DB"."MODE BUFF", in2 := 1)
      { S7_Templates := "SrcType := Int" } NE_Contact(in1 := "CONTINUE DB"."PREMIXING PROCESS ERROR", in2 := 1)
      Coil( "AUTO SUBOUTPUT DB"."PBV-15 VACUUM INLET" )
   END_RUNG
   // the same network as SCL:
   "AUTO SUBOUTPUT DB"."PBV-15 VACUUM INLET" := "AlwaysTRUE" AND ("MODE SELECTION DB"."MODE BUFF" = 1) AND ("CONTINUE DB"."PREMIXING PROCESS ERROR" <> 1);
END_REGION

REGION Network 25: PBV-16 VACUUM VENT VALVE
   RUNG wire#powerrail
      Contact( "AlwaysFALSE" )
      { S7_Templates := "SrcType := Int" } EQ_Contact(in1 := "MODE SELECTION DB"."MODE BUFF", in2 := 1)
      Coil( "AUTO SUBOUTPUT DB"."PBV-16 VACUUM VENT VALVE" )
   END_RUNG
   // the same network as SCL:
   "AUTO SUBOUTPUT DB"."PBV-16 VACUUM VENT VALVE" := "AlwaysFALSE" AND ("MODE SELECTION DB"."MODE BUFF" = 1);
END_REGION

REGION Network 26: PFBV-17 TANK OUTLET VALVE
   RUNG wire#powerrail
      Contact( "AlwaysTRUE" )
      { S7_Templates := "SrcType := Int" } EQ_Contact(in1 := "MODE SELECTION DB"."MODE BUFF", in2 := 1)
      I_Contact( "PREMIXING DB".PAUSE )
      { S7_Templates := "SrcType := Int" } EQ_Contact(in1 := "PREMIXING DB"."AUTO BUFF", in2 := 160)
      { S7_Templates := "SrcType := Int" } NE_Contact(in1 := "CONTINUE DB"."PREMIXING PROCESS ERROR", in2 := 1)
      Coil( "AUTO SUBOUTPUT DB"."PFBV-17 TANK OUTLET VALVE" )
   END_RUNG
   // the same network as SCL:
   "AUTO SUBOUTPUT DB"."PFBV-17 TANK OUTLET VALVE" := "AlwaysTRUE" AND ("MODE SELECTION DB"."MODE BUFF" = 1) AND NOT "PREMIXING DB".PAUSE AND ("PREMIXING DB"."AUTO BUFF" = 160) AND ("CONTINUE DB"."PREMIXING PROCESS ERROR" <> 1);
END_REGION

REGION Network 27: PBV-19 PW INLET
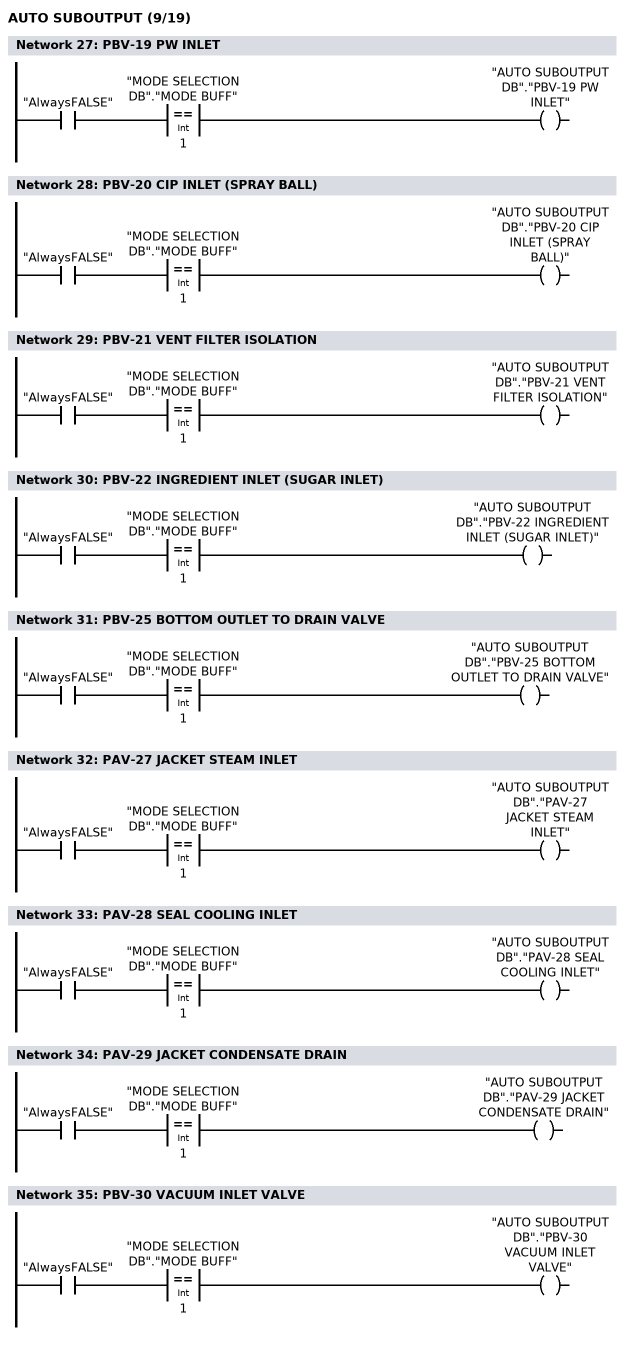
   RUNG wire#powerrail
      Contact( "AlwaysFALSE" )
      { S7_Templates := "SrcType := Int" } EQ_Contact(in1 := "MODE SELECTION DB"."MODE BUFF", in2 := 1)
      Coil( "AUTO SUBOUTPUT DB"."PBV-19 PW INLET" )
   END_RUNG
   // the same network as SCL:
   "AUTO SUBOUTPUT DB"."PBV-19 PW INLET" := "AlwaysFALSE" AND ("MODE SELECTION DB"."MODE BUFF" = 1);
END_REGION

REGION Network 28: PBV-20 CIP INLET (SPRAY BALL)
   RUNG wire#powerrail
      Contact( "AlwaysFALSE" )
      { S7_Templates := "SrcType := Int" } EQ_Contact(in1 := "MODE SELECTION DB"."MODE BUFF", in2 := 1)
      Coil( "AUTO SUBOUTPUT DB"."PBV-20 CIP INLET (SPRAY BALL)" )
   END_RUNG
   // the same network as SCL:
   "AUTO SUBOUTPUT DB"."PBV-20 CIP INLET (SPRAY BALL)" := "AlwaysFALSE" AND ("MODE SELECTION DB"."MODE BUFF" = 1);
END_REGION

REGION Network 29: PBV-21 VENT FILTER ISOLATION
   RUNG wire#powerrail
      Contact( "AlwaysFALSE" )
      { S7_Templates := "SrcType := Int" } EQ_Contact(in1 := "MODE SELECTION DB"."MODE BUFF", in2 := 1)
      Coil( "AUTO SUBOUTPUT DB"."PBV-21 VENT FILTER ISOLATION" )
   END_RUNG
   // the same network as SCL:
   "AUTO SUBOUTPUT DB"."PBV-21 VENT FILTER ISOLATION" := "AlwaysFALSE" AND ("MODE SELECTION DB"."MODE BUFF" = 1);
END_REGION

REGION Network 30: PBV-22 INGREDIENT INLET (SUGAR INLET)
   RUNG wire#powerrail
      Contact( "AlwaysFALSE" )
      { S7_Templates := "SrcType := Int" } EQ_Contact(in1 := "MODE SELECTION DB"."MODE BUFF", in2 := 1)
      Coil( "AUTO SUBOUTPUT DB"."PBV-22 INGREDIENT INLET (SUGAR INLET)" )
   END_RUNG
   // the same network as SCL:
   "AUTO SUBOUTPUT DB"."PBV-22 INGREDIENT INLET (SUGAR INLET)" := "AlwaysFALSE" AND ("MODE SELECTION DB"."MODE BUFF" = 1);
END_REGION

REGION Network 31: PBV-25 BOTTOM OUTLET TO DRAIN VALVE
   RUNG wire#powerrail
      Contact( "AlwaysFALSE" )
      { S7_Templates := "SrcType := Int" } EQ_Contact(in1 := "MODE SELECTION DB"."MODE BUFF", in2 := 1)
      Coil( "AUTO SUBOUTPUT DB"."PBV-25 BOTTOM OUTLET TO DRAIN VALVE" )
   END_RUNG
   // the same network as SCL:
   "AUTO SUBOUTPUT DB"."PBV-25 BOTTOM OUTLET TO DRAIN VALVE" := "AlwaysFALSE" AND ("MODE SELECTION DB"."MODE BUFF" = 1);
END_REGION

REGION Network 32: PAV-27 JACKET STEAM INLET
   RUNG wire#powerrail
      Contact( "AlwaysFALSE" )
      { S7_Templates := "SrcType := Int" } EQ_Contact(in1 := "MODE SELECTION DB"."MODE BUFF", in2 := 1)
      Coil( "AUTO SUBOUTPUT DB"."PAV-27 JACKET STEAM INLET" )
   END_RUNG
   // the same network as SCL:
   "AUTO SUBOUTPUT DB"."PAV-27 JACKET STEAM INLET" := "AlwaysFALSE" AND ("MODE SELECTION DB"."MODE BUFF" = 1);
END_REGION

REGION Network 33: PAV-28 SEAL COOLING INLET
   RUNG wire#powerrail
      Contact( "AlwaysFALSE" )
      { S7_Templates := "SrcType := Int" } EQ_Contact(in1 := "MODE SELECTION DB"."MODE BUFF", in2 := 1)
      Coil( "AUTO SUBOUTPUT DB"."PAV-28 SEAL COOLING INLET" )
   END_RUNG
   // the same network as SCL:
   "AUTO SUBOUTPUT DB"."PAV-28 SEAL COOLING INLET" := "AlwaysFALSE" AND ("MODE SELECTION DB"."MODE BUFF" = 1);
END_REGION

REGION Network 34: PAV-29 JACKET CONDENSATE DRAIN
   RUNG wire#powerrail
      Contact( "AlwaysFALSE" )
      { S7_Templates := "SrcType := Int" } EQ_Contact(in1 := "MODE SELECTION DB"."MODE BUFF", in2 := 1)
      Coil( "AUTO SUBOUTPUT DB"."PAV-29 JACKET CONDENSATE DRAIN" )
   END_RUNG
   // the same network as SCL:
   "AUTO SUBOUTPUT DB"."PAV-29 JACKET CONDENSATE DRAIN" := "AlwaysFALSE" AND ("MODE SELECTION DB"."MODE BUFF" = 1);
END_REGION

REGION Network 35: PBV-30 VACUUM INLET VALVE
   RUNG wire#powerrail
      Contact( "AlwaysFALSE" )
      { S7_Templates := "SrcType := Int" } EQ_Contact(in1 := "MODE SELECTION DB"."MODE BUFF", in2 := 1)
      Coil( "AUTO SUBOUTPUT DB"."PBV-30 VACUUM INLET VALVE" )
   END_RUNG
   // the same network as SCL:
   "AUTO SUBOUTPUT DB"."PBV-30 VACUUM INLET VALVE" := "AlwaysFALSE" AND ("MODE SELECTION DB"."MODE BUFF" = 1);
END_REGION

REGION Network 36: PBV-31 VACUUM VENT VALVE
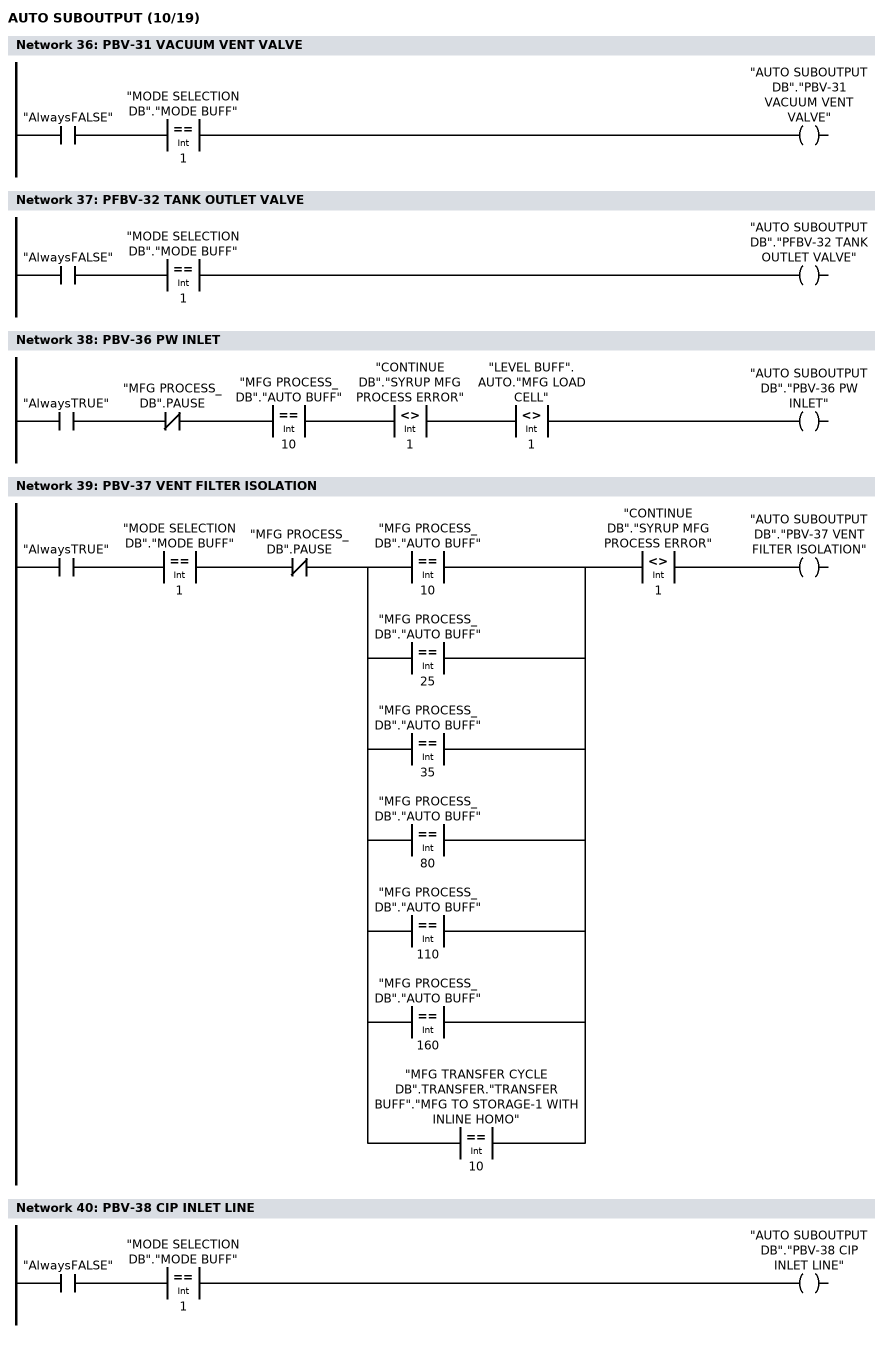
   RUNG wire#powerrail
      Contact( "AlwaysFALSE" )
      { S7_Templates := "SrcType := Int" } EQ_Contact(in1 := "MODE SELECTION DB"."MODE BUFF", in2 := 1)
      Coil( "AUTO SUBOUTPUT DB"."PBV-31 VACUUM VENT VALVE" )
   END_RUNG
   // the same network as SCL:
   "AUTO SUBOUTPUT DB"."PBV-31 VACUUM VENT VALVE" := "AlwaysFALSE" AND ("MODE SELECTION DB"."MODE BUFF" = 1);
END_REGION

REGION Network 37: PFBV-32 TANK OUTLET VALVE
   RUNG wire#powerrail
      Contact( "AlwaysFALSE" )
      { S7_Templates := "SrcType := Int" } EQ_Contact(in1 := "MODE SELECTION DB"."MODE BUFF", in2 := 1)
      Coil( "AUTO SUBOUTPUT DB"."PFBV-32 TANK OUTLET VALVE" )
   END_RUNG
   // the same network as SCL:
   "AUTO SUBOUTPUT DB"."PFBV-32 TANK OUTLET VALVE" := "AlwaysFALSE" AND ("MODE SELECTION DB"."MODE BUFF" = 1);
END_REGION

REGION Network 38: PBV-36 PW INLET
   RUNG wire#powerrail
      Contact( "AlwaysTRUE" )
      I_Contact( "MFG PROCESS_DB".PAUSE )
      { S7_Templates := "SrcType := Int" } EQ_Contact(in1 := "MFG PROCESS_DB"."AUTO BUFF", in2 := 10)
      { S7_Templates := "SrcType := Int" } NE_Contact(in1 := "CONTINUE DB"."SYRUP MFG PROCESS ERROR", in2 := 1)
      { S7_Templates := "SrcType := Int" } NE_Contact(in1 := "LEVEL BUFF".AUTO."MFG LOAD CELL", in2 := 1)
      Coil( "AUTO SUBOUTPUT DB"."PBV-36 PW INLET" )
   END_RUNG
   // the same network as SCL:
   "AUTO SUBOUTPUT DB"."PBV-36 PW INLET" := "AlwaysTRUE" AND NOT "MFG PROCESS_DB".PAUSE AND ("MFG PROCESS_DB"."AUTO BUFF" = 10) AND ("CONTINUE DB"."SYRUP MFG PROCESS ERROR" <> 1) AND ("LEVEL BUFF".AUTO."MFG LOAD CELL" <> 1);
END_REGION

REGION Network 39: PBV-37 VENT FILTER ISOLATION
   RUNG wire#powerrail
      Contact( "AlwaysTRUE" )
      { S7_Templates := "SrcType := Int" } EQ_Contact(in1 := "MODE SELECTION DB"."MODE BUFF", in2 := 1)
      I_Contact( "MFG PROCESS_DB".PAUSE )
      wire#w1
      { S7_Templates := "SrcType := Int" } EQ_Contact(in1 := "MFG PROCESS_DB"."AUTO BUFF", in2 := 10)
      wire#w2
      { S7_Templates := "SrcType := Int" } NE_Contact(in1 := "CONTINUE DB"."SYRUP MFG PROCESS ERROR", in2 := 1)
      Coil( "AUTO SUBOUTPUT DB"."PBV-37 VENT FILTER ISOLATION" )
   END_RUNG
   RUNG wire#w1
      { S7_Templates := "SrcType := Int" } EQ_Contact(in1 := "MFG PROCESS_DB"."AUTO BUFF", in2 := 25)
   END_RUNG wire#w2
   RUNG wire#w1
      { S7_Templates := "SrcType := Int" } EQ_Contact(in1 := "MFG PROCESS_DB"."AUTO BUFF", in2 := 35)
   END_RUNG wire#w2
   RUNG wire#w1
      { S7_Templates := "SrcType := Int" } EQ_Contact(in1 := "MFG PROCESS_DB"."AUTO BUFF", in2 := 80)
   END_RUNG wire#w2
   RUNG wire#w1
      { S7_Templates := "SrcType := Int" } EQ_Contact(in1 := "MFG PROCESS_DB"."AUTO BUFF", in2 := 110)
   END_RUNG wire#w2
   RUNG wire#w1
      { S7_Templates := "SrcType := Int" } EQ_Contact(in1 := "MFG PROCESS_DB"."AUTO BUFF", in2 := 160)
   END_RUNG wire#w2
   RUNG wire#w1
      { S7_Templates := "SrcType := Int" } EQ_Contact(in1 := "MFG TRANSFER CYCLE DB".TRANSFER."TRANSFER BUFF"."MFG TO STORAGE-1 WITH INLINE HOMO", in2 := 10)
   END_RUNG wire#w2
   // the same network as SCL:
   "AUTO SUBOUTPUT DB"."PBV-37 VENT FILTER ISOLATION" := "AlwaysTRUE" AND ("MODE SELECTION DB"."MODE BUFF" = 1) AND NOT "MFG PROCESS_DB".PAUSE AND (("MFG PROCESS_DB"."AUTO BUFF" = 10) OR ("MFG PROCESS_DB"."AUTO BUFF" = 25) OR ("MFG PROCESS_DB"."AUTO BUFF" = 35) OR ("MFG PROCESS_DB"."AUTO BUFF" = 80) OR ("MFG PROCESS_DB"."AUTO BUFF" = 110) OR ("MFG PROCESS_DB"."AUTO BUFF" = 160) OR ("MFG TRANSFER CYCLE DB".TRANSFER."TRANSFER BUFF"."MFG TO STORAGE-1 WITH INLINE HOMO" = 10)) AND ("CONTINUE DB"."SYRUP MFG PROCESS ERROR" <> 1);
END_REGION

REGION Network 40: PBV-38 CIP INLET LINE
   RUNG wire#powerrail
      Contact( "AlwaysFALSE" )
      { S7_Templates := "SrcType := Int" } EQ_Contact(in1 := "MODE SELECTION DB"."MODE BUFF", in2 := 1)
      Coil( "AUTO SUBOUTPUT DB"."PBV-38 CIP INLET LINE" )
   END_RUNG
   // the same network as SCL:
   "AUTO SUBOUTPUT DB"."PBV-38 CIP INLET LINE" := "AlwaysFALSE" AND ("MODE SELECTION DB"."MODE BUFF" = 1);
END_REGION

REGION Network 41: PBV-41 MFG TANK DRAIN VALVE
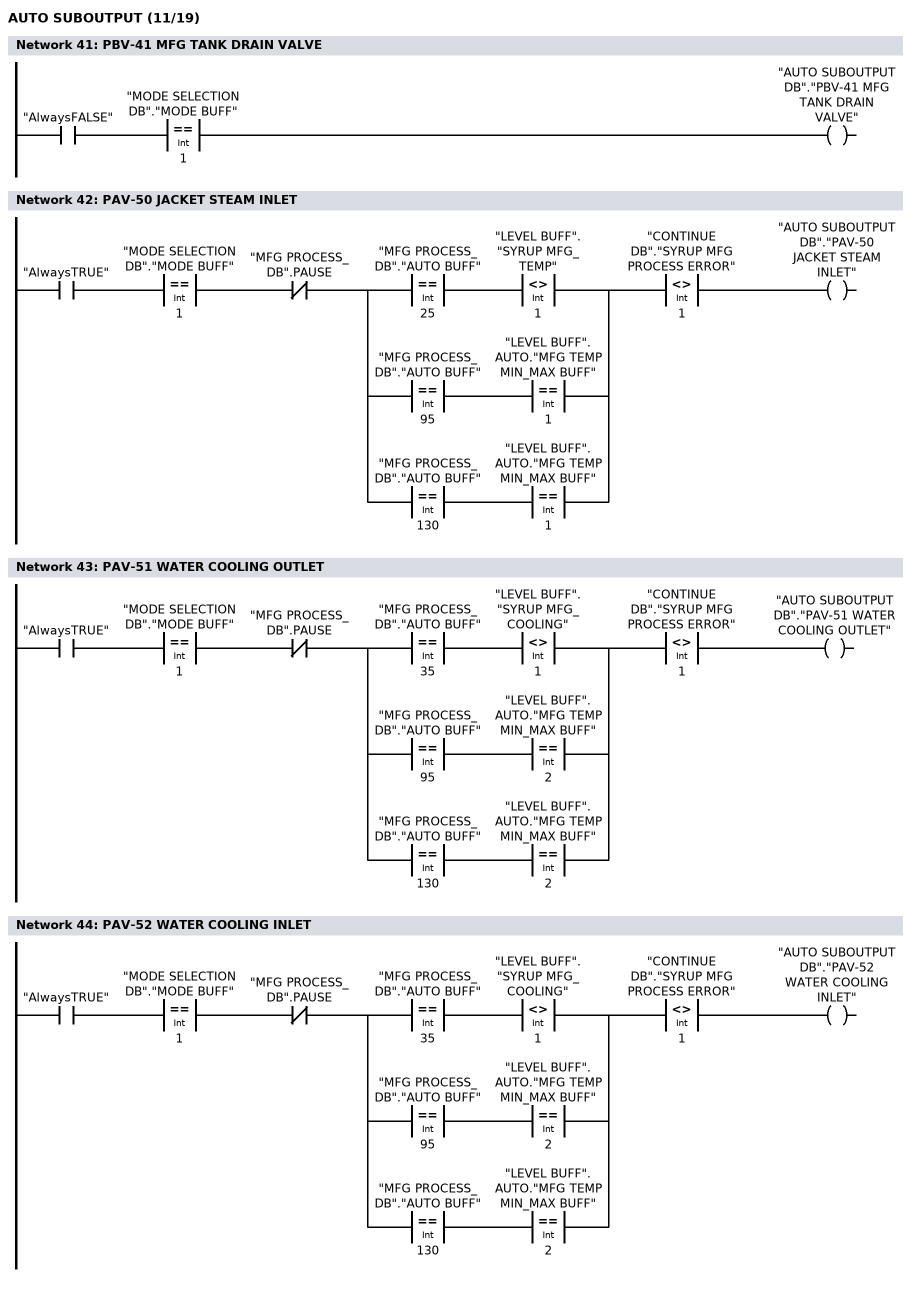
   RUNG wire#powerrail
      Contact( "AlwaysFALSE" )
      { S7_Templates := "SrcType := Int" } EQ_Contact(in1 := "MODE SELECTION DB"."MODE BUFF", in2 := 1)
      Coil( "AUTO SUBOUTPUT DB"."PBV-41 MFG TANK DRAIN VALVE" )
   END_RUNG
   // the same network as SCL:
   "AUTO SUBOUTPUT DB"."PBV-41 MFG TANK DRAIN VALVE" := "AlwaysFALSE" AND ("MODE SELECTION DB"."MODE BUFF" = 1);
END_REGION

REGION Network 42: PAV-50 JACKET STEAM INLET
   RUNG wire#powerrail
      Contact( "AlwaysTRUE" )
      { S7_Templates := "SrcType := Int" } EQ_Contact(in1 := "MODE SELECTION DB"."MODE BUFF", in2 := 1)
      I_Contact( "MFG PROCESS_DB".PAUSE )
      wire#w1
      { S7_Templates := "SrcType := Int" } EQ_Contact(in1 := "MFG PROCESS_DB"."AUTO BUFF", in2 := 25)
      { S7_Templates := "SrcType := Int" } NE_Contact(in1 := "LEVEL BUFF"."SYRUP MFG_TEMP", in2 := 1)
      wire#w2
      { S7_Templates := "SrcType := Int" } NE_Contact(in1 := "CONTINUE DB"."SYRUP MFG PROCESS ERROR", in2 := 1)
      Coil( "AUTO SUBOUTPUT DB"."PAV-50 JACKET STEAM INLET" )
   END_RUNG
   RUNG wire#w1
      { S7_Templates := "SrcType := Int" } EQ_Contact(in1 := "MFG PROCESS_DB"."AUTO BUFF", in2 := 95)
      { S7_Templates := "SrcType := Int" } EQ_Contact(in1 := "LEVEL BUFF".AUTO."MFG TEMP MIN_MAX BUFF", in2 := 1)
   END_RUNG wire#w2
   RUNG wire#w1
      { S7_Templates := "SrcType := Int" } EQ_Contact(in1 := "MFG PROCESS_DB"."AUTO BUFF", in2 := 130)
      { S7_Templates := "SrcType := Int" } EQ_Contact(in1 := "LEVEL BUFF".AUTO."MFG TEMP MIN_MAX BUFF", in2 := 1)
   END_RUNG wire#w2
   // the same network as SCL:
   "AUTO SUBOUTPUT DB"."PAV-50 JACKET STEAM INLET" := "AlwaysTRUE" AND ("MODE SELECTION DB"."MODE BUFF" = 1) AND NOT "MFG PROCESS_DB".PAUSE AND ((("MFG PROCESS_DB"."AUTO BUFF" = 25) AND ("LEVEL BUFF"."SYRUP MFG_TEMP" <> 1)) OR (("MFG PROCESS_DB"."AUTO BUFF" = 95) AND ("LEVEL BUFF".AUTO."MFG TEMP MIN_MAX BUFF" = 1)) OR (("MFG PROCESS_DB"."AUTO BUFF" = 130) AND ("LEVEL BUFF".AUTO."MFG TEMP MIN_MAX BUFF" = 1))) AND ("CONTINUE DB"."SYRUP MFG PROCESS ERROR" <> 1);
END_REGION

REGION Network 43: PAV-51 WATER COOLING OUTLET
   RUNG wire#powerrail
      Contact( "AlwaysTRUE" )
      { S7_Templates := "SrcType := Int" } EQ_Contact(in1 := "MODE SELECTION DB"."MODE BUFF", in2 := 1)
      I_Contact( "MFG PROCESS_DB".PAUSE )
      wire#w1
      { S7_Templates := "SrcType := Int" } EQ_Contact(in1 := "MFG PROCESS_DB"."AUTO BUFF", in2 := 35)
      { S7_Templates := "SrcType := Int" } NE_Contact(in1 := "LEVEL BUFF"."SYRUP MFG_COOLING", in2 := 1)
      wire#w2
      { S7_Templates := "SrcType := Int" } NE_Contact(in1 := "CONTINUE DB"."SYRUP MFG PROCESS ERROR", in2 := 1)
      Coil( "AUTO SUBOUTPUT DB"."PAV-51 WATER COOLING OUTLET" )
   END_RUNG
   RUNG wire#w1
      { S7_Templates := "SrcType := Int" } EQ_Contact(in1 := "MFG PROCESS_DB"."AUTO BUFF", in2 := 95)
      { S7_Templates := "SrcType := Int" } EQ_Contact(in1 := "LEVEL BUFF".AUTO."MFG TEMP MIN_MAX BUFF", in2 := 2)
   END_RUNG wire#w2
   RUNG wire#w1
      { S7_Templates := "SrcType := Int" } EQ_Contact(in1 := "MFG PROCESS_DB"."AUTO BUFF", in2 := 130)
      { S7_Templates := "SrcType := Int" } EQ_Contact(in1 := "LEVEL BUFF".AUTO."MFG TEMP MIN_MAX BUFF", in2 := 2)
   END_RUNG wire#w2
   // the same network as SCL:
   "AUTO SUBOUTPUT DB"."PAV-51 WATER COOLING OUTLET" := "AlwaysTRUE" AND ("MODE SELECTION DB"."MODE BUFF" = 1) AND NOT "MFG PROCESS_DB".PAUSE AND ((("MFG PROCESS_DB"."AUTO BUFF" = 35) AND ("LEVEL BUFF"."SYRUP MFG_COOLING" <> 1)) OR (("MFG PROCESS_DB"."AUTO BUFF" = 95) AND ("LEVEL BUFF".AUTO."MFG TEMP MIN_MAX BUFF" = 2)) OR (("MFG PROCESS_DB"."AUTO BUFF" = 130) AND ("LEVEL BUFF".AUTO."MFG TEMP MIN_MAX BUFF" = 2))) AND ("CONTINUE DB"."SYRUP MFG PROCESS ERROR" <> 1);
END_REGION

REGION Network 44: PAV-52 WATER COOLING INLET
   RUNG wire#powerrail
      Contact( "AlwaysTRUE" )
      { S7_Templates := "SrcType := Int" } EQ_Contact(in1 := "MODE SELECTION DB"."MODE BUFF", in2 := 1)
      I_Contact( "MFG PROCESS_DB".PAUSE )
      wire#w1
      { S7_Templates := "SrcType := Int" } EQ_Contact(in1 := "MFG PROCESS_DB"."AUTO BUFF", in2 := 35)
      { S7_Templates := "SrcType := Int" } NE_Contact(in1 := "LEVEL BUFF"."SYRUP MFG_COOLING", in2 := 1)
      wire#w2
      { S7_Templates := "SrcType := Int" } NE_Contact(in1 := "CONTINUE DB"."SYRUP MFG PROCESS ERROR", in2 := 1)
      Coil( "AUTO SUBOUTPUT DB"."PAV-52 WATER COOLING INLET" )
   END_RUNG
   RUNG wire#w1
      { S7_Templates := "SrcType := Int" } EQ_Contact(in1 := "MFG PROCESS_DB"."AUTO BUFF", in2 := 95)
      { S7_Templates := "SrcType := Int" } EQ_Contact(in1 := "LEVEL BUFF".AUTO."MFG TEMP MIN_MAX BUFF", in2 := 2)
   END_RUNG wire#w2
   RUNG wire#w1
      { S7_Templates := "SrcType := Int" } EQ_Contact(in1 := "MFG PROCESS_DB"."AUTO BUFF", in2 := 130)
      { S7_Templates := "SrcType := Int" } EQ_Contact(in1 := "LEVEL BUFF".AUTO."MFG TEMP MIN_MAX BUFF", in2 := 2)
   END_RUNG wire#w2
   // the same network as SCL:
   "AUTO SUBOUTPUT DB"."PAV-52 WATER COOLING INLET" := "AlwaysTRUE" AND ("MODE SELECTION DB"."MODE BUFF" = 1) AND NOT "MFG PROCESS_DB".PAUSE AND ((("MFG PROCESS_DB"."AUTO BUFF" = 35) AND ("LEVEL BUFF"."SYRUP MFG_COOLING" <> 1)) OR (("MFG PROCESS_DB"."AUTO BUFF" = 95) AND ("LEVEL BUFF".AUTO."MFG TEMP MIN_MAX BUFF" = 2)) OR (("MFG PROCESS_DB"."AUTO BUFF" = 130) AND ("LEVEL BUFF".AUTO."MFG TEMP MIN_MAX BUFF" = 2))) AND ("CONTINUE DB"."SYRUP MFG PROCESS ERROR" <> 1);
END_REGION

REGION Network 45: PAV-53 SEAL COOLING INLET
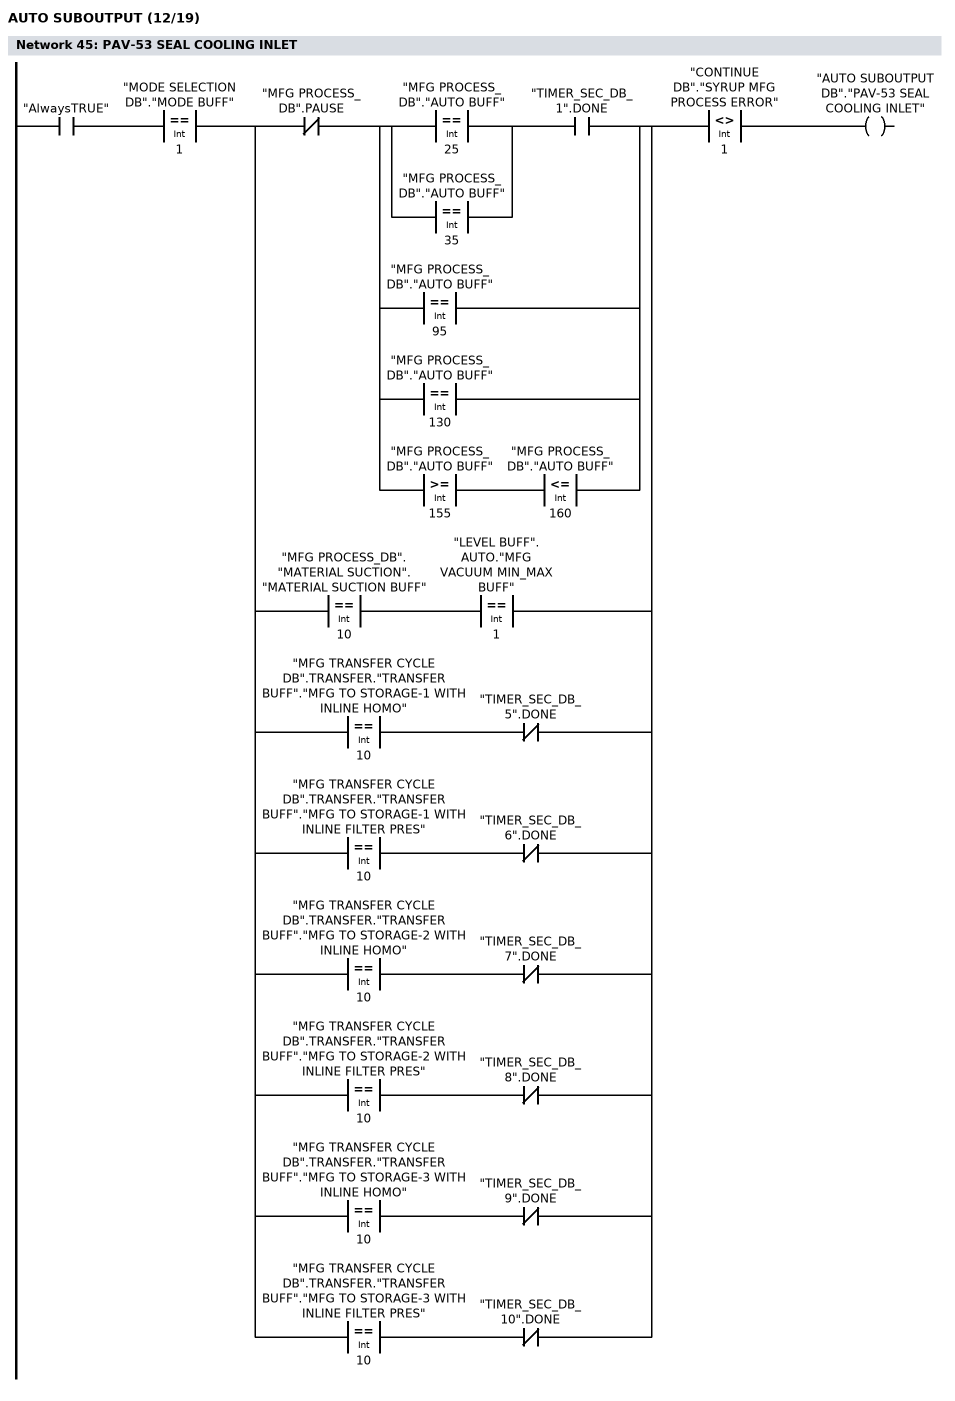
   RUNG wire#powerrail
      Contact( "AlwaysTRUE" )
      { S7_Templates := "SrcType := Int" } EQ_Contact(in1 := "MODE SELECTION DB"."MODE BUFF", in2 := 1)
      wire#w1
      I_Contact( "MFG PROCESS_DB".PAUSE )
      wire#w2
      { S7_Templates := "SrcType := Int" } EQ_Contact(in1 := "MFG PROCESS_DB"."AUTO BUFF", in2 := 25)
      wire#w3
      Contact( "TIMER_SEC_DB_1".DONE )
      wire#w4
      { S7_Templates := "SrcType := Int" } NE_Contact(in1 := "CONTINUE DB"."SYRUP MFG PROCESS ERROR", in2 := 1)
      Coil( "AUTO SUBOUTPUT DB"."PAV-53 SEAL COOLING INLET" )
   END_RUNG
   RUNG wire#w2
      { S7_Templates := "SrcType := Int" } EQ_Contact(in1 := "MFG PROCESS_DB"."AUTO BUFF", in2 := 35)
   END_RUNG wire#w3
   RUNG wire#w2
      { S7_Templates := "SrcType := Int" } EQ_Contact(in1 := "MFG PROCESS_DB"."AUTO BUFF", in2 := 95)
   END_RUNG wire#w4
   RUNG wire#w2
      { S7_Templates := "SrcType := Int" } EQ_Contact(in1 := "MFG PROCESS_DB"."AUTO BUFF", in2 := 130)
   END_RUNG wire#w4
   RUNG wire#w2
      { S7_Templates := "SrcType := Int" } GE_Contact(in1 := "MFG PROCESS_DB"."AUTO BUFF", in2 := 155)
      { S7_Templates := "SrcType := Int" } LE_Contact(in1 := "MFG PROCESS_DB"."AUTO BUFF", in2 := 160)
   END_RUNG wire#w4
   RUNG wire#w1
      { S7_Templates := "SrcType := Int" } EQ_Contact(in1 := "MFG PROCESS_DB"."MATERIAL SUCTION"."MATERIAL SUCTION BUFF", in2 := 10)
      { S7_Templates := "SrcType := Int" } EQ_Contact(in1 := "LEVEL BUFF".AUTO."MFG VACUUM MIN_MAX BUFF", in2 := 1)
   END_RUNG wire#w4
   RUNG wire#w1
      { S7_Templates := "SrcType := Int" } EQ_Contact(in1 := "MFG TRANSFER CYCLE DB".TRANSFER."TRANSFER BUFF"."MFG TO STORAGE-1 WITH INLINE HOMO", in2 := 10)
      I_Contact( "TIMER_SEC_DB_5".DONE )
   END_RUNG wire#w4
   RUNG wire#w1
      { S7_Templates := "SrcType := Int" } EQ_Contact(in1 := "MFG TRANSFER CYCLE DB".TRANSFER."TRANSFER BUFF"."MFG TO STORAGE-1 WITH INLINE FILTER PRES", in2 := 10)
      I_Contact( "TIMER_SEC_DB_6".DONE )
   END_RUNG wire#w4
   RUNG wire#w1
      { S7_Templates := "SrcType := Int" } EQ_Contact(in1 := "MFG TRANSFER CYCLE DB".TRANSFER."TRANSFER BUFF"."MFG TO STORAGE-2 WITH INLINE HOMO", in2 := 10)
      I_Contact( "TIMER_SEC_DB_7".DONE )
   END_RUNG wire#w4
   RUNG wire#w1
      { S7_Templates := "SrcType := Int" } EQ_Contact(in1 := "MFG TRANSFER CYCLE DB".TRANSFER."TRANSFER BUFF"."MFG TO STORAGE-2 WITH INLINE FILTER PRES", in2 := 10)
      I_Contact( "TIMER_SEC_DB_8".DONE )
   END_RUNG wire#w4
   RUNG wire#w1
      { S7_Templates := "SrcType := Int" } EQ_Contact(in1 := "MFG TRANSFER CYCLE DB".TRANSFER."TRANSFER BUFF"."MFG TO STORAGE-3 WITH INLINE HOMO", in2 := 10)
      I_Contact( "TIMER_SEC_DB_9".DONE )
   END_RUNG wire#w4
   RUNG wire#w1
      { S7_Templates := "SrcType := Int" } EQ_Contact(in1 := "MFG TRANSFER CYCLE DB".TRANSFER."TRANSFER BUFF"."MFG TO STORAGE-3 WITH INLINE FILTER PRES", in2 := 10)
      I_Contact( "TIMER_SEC_DB_10".DONE )
   END_RUNG wire#w4
   // the same network as SCL:
   "AUTO SUBOUTPUT DB"."PAV-53 SEAL COOLING INLET" := "AlwaysTRUE" AND ("MODE SELECTION DB"."MODE BUFF" = 1) AND ((NOT "MFG PROCESS_DB".PAUSE AND (((("MFG PROCESS_DB"."AUTO BUFF" = 25) OR ("MFG PROCESS_DB"."AUTO BUFF" = 35)) AND "TIMER_SEC_DB_1".DONE) OR ("MFG PROCESS_DB"."AUTO BUFF" = 95) OR ("MFG PROCESS_DB"."AUTO BUFF" = 130) OR (("MFG PROCESS_DB"."AUTO BUFF" >= 155) AND ("MFG PROCESS_DB"."AUTO BUFF" <= 160)))) OR (("MFG PROCESS_DB"."MATERIAL SUCTION"."MATERIAL SUCTION BUFF" = 10) AND ("LEVEL BUFF".AUTO."MFG VACUUM MIN_MAX BUFF" = 1)) OR (("MFG TRANSFER CYCLE DB".TRANSFER."TRANSFER BUFF"."MFG TO STORAGE-1 WITH INLINE HOMO" = 10) AND NOT "TIMER_SEC_DB_5".DONE) OR (("MFG TRANSFER CYCLE DB".TRANSFER."TRANSFER BUFF"."MFG TO STORAGE-1 WITH INLINE FILTER PRES" = 10) AND NOT "TIMER_SEC_DB_6".DONE) OR (("MFG TRANSFER CYCLE DB".TRANSFER."TRANSFER BUFF"."MFG TO STORAGE-2 WITH INLINE HOMO" = 10) AND NOT "TIMER_SEC_DB_7".DONE) OR (("MFG TRANSFER CYCLE DB".TRANSFER."TRANSFER BUFF"."MFG TO STORAGE-2 WITH INLINE FILTER PRES" = 10) AND NOT "TIMER_SEC_DB_8".DONE) OR (("MFG TRANSFER CYCLE DB".TRANSFER."TRANSFER BUFF"."MFG TO STORAGE-3 WITH INLINE HOMO" = 10) AND NOT "TIMER_SEC_DB_9".DONE) OR (("MFG TRANSFER CYCLE DB".TRANSFER."TRANSFER BUFF"."MFG TO STORAGE-3 WITH INLINE FILTER PRES" = 10) AND NOT "TIMER_SEC_DB_10".DONE)) AND ("CONTINUE DB"."SYRUP MFG PROCESS ERROR" <> 1);
END_REGION

REGION Network 46: PAV-54 JACKET STEAM OUTLET VALVE
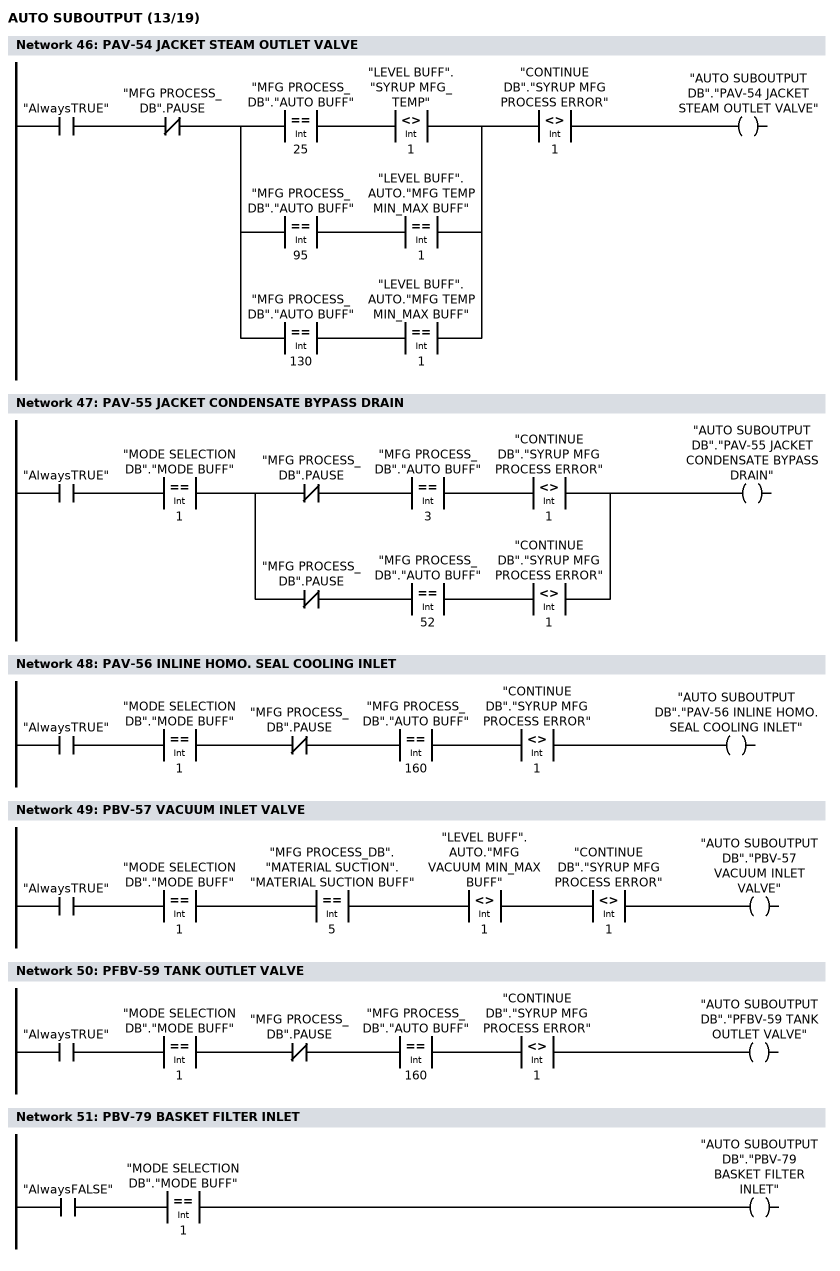
   RUNG wire#powerrail
      Contact( "AlwaysTRUE" )
      I_Contact( "MFG PROCESS_DB".PAUSE )
      wire#w1
      { S7_Templates := "SrcType := Int" } EQ_Contact(in1 := "MFG PROCESS_DB"."AUTO BUFF", in2 := 25)
      { S7_Templates := "SrcType := Int" } NE_Contact(in1 := "LEVEL BUFF"."SYRUP MFG_TEMP", in2 := 1)
      wire#w2
      { S7_Templates := "SrcType := Int" } NE_Contact(in1 := "CONTINUE DB"."SYRUP MFG PROCESS ERROR", in2 := 1)
      Coil( "AUTO SUBOUTPUT DB"."PAV-54 JACKET STEAM OUTLET VALVE" )
   END_RUNG
   RUNG wire#w1
      { S7_Templates := "SrcType := Int" } EQ_Contact(in1 := "MFG PROCESS_DB"."AUTO BUFF", in2 := 95)
      { S7_Templates := "SrcType := Int" } EQ_Contact(in1 := "LEVEL BUFF".AUTO."MFG TEMP MIN_MAX BUFF", in2 := 1)
   END_RUNG wire#w2
   RUNG wire#w1
      { S7_Templates := "SrcType := Int" } EQ_Contact(in1 := "MFG PROCESS_DB"."AUTO BUFF", in2 := 130)
      { S7_Templates := "SrcType := Int" } EQ_Contact(in1 := "LEVEL BUFF".AUTO."MFG TEMP MIN_MAX BUFF", in2 := 1)
   END_RUNG wire#w2
   // the same network as SCL:
   "AUTO SUBOUTPUT DB"."PAV-54 JACKET STEAM OUTLET VALVE" := "AlwaysTRUE" AND NOT "MFG PROCESS_DB".PAUSE AND ((("MFG PROCESS_DB"."AUTO BUFF" = 25) AND ("LEVEL BUFF"."SYRUP MFG_TEMP" <> 1)) OR (("MFG PROCESS_DB"."AUTO BUFF" = 95) AND ("LEVEL BUFF".AUTO."MFG TEMP MIN_MAX BUFF" = 1)) OR (("MFG PROCESS_DB"."AUTO BUFF" = 130) AND ("LEVEL BUFF".AUTO."MFG TEMP MIN_MAX BUFF" = 1))) AND ("CONTINUE DB"."SYRUP MFG PROCESS ERROR" <> 1);
END_REGION

REGION Network 47: PAV-55 JACKET CONDENSATE BYPASS DRAIN
   RUNG wire#powerrail
      Contact( "AlwaysTRUE" )
      { S7_Templates := "SrcType := Int" } EQ_Contact(in1 := "MODE SELECTION DB"."MODE BUFF", in2 := 1)
      wire#w1
      I_Contact( "MFG PROCESS_DB".PAUSE )
      { S7_Templates := "SrcType := Int" } EQ_Contact(in1 := "MFG PROCESS_DB"."AUTO BUFF", in2 := 3)
      { S7_Templates := "SrcType := Int" } NE_Contact(in1 := "CONTINUE DB"."SYRUP MFG PROCESS ERROR", in2 := 1)
      wire#w2
      Coil( "AUTO SUBOUTPUT DB"."PAV-55 JACKET CONDENSATE BYPASS DRAIN" )
   END_RUNG
   RUNG wire#w1
      I_Contact( "MFG PROCESS_DB".PAUSE )
      { S7_Templates := "SrcType := Int" } EQ_Contact(in1 := "MFG PROCESS_DB"."AUTO BUFF", in2 := 52)
      { S7_Templates := "SrcType := Int" } NE_Contact(in1 := "CONTINUE DB"."SYRUP MFG PROCESS ERROR", in2 := 1)
   END_RUNG wire#w2
   // the same network as SCL:
   "AUTO SUBOUTPUT DB"."PAV-55 JACKET CONDENSATE BYPASS DRAIN" := "AlwaysTRUE" AND ("MODE SELECTION DB"."MODE BUFF" = 1) AND ((NOT "MFG PROCESS_DB".PAUSE AND ("MFG PROCESS_DB"."AUTO BUFF" = 3) AND ("CONTINUE DB"."SYRUP MFG PROCESS ERROR" <> 1)) OR (NOT "MFG PROCESS_DB".PAUSE AND ("MFG PROCESS_DB"."AUTO BUFF" = 52) AND ("CONTINUE DB"."SYRUP MFG PROCESS ERROR" <> 1)));
END_REGION

REGION Network 48: PAV-56 INLINE HOMO. SEAL COOLING INLET
   RUNG wire#powerrail
      Contact( "AlwaysTRUE" )
      { S7_Templates := "SrcType := Int" } EQ_Contact(in1 := "MODE SELECTION DB"."MODE BUFF", in2 := 1)
      I_Contact( "MFG PROCESS_DB".PAUSE )
      { S7_Templates := "SrcType := Int" } EQ_Contact(in1 := "MFG PROCESS_DB"."AUTO BUFF", in2 := 160)
      { S7_Templates := "SrcType := Int" } NE_Contact(in1 := "CONTINUE DB"."SYRUP MFG PROCESS ERROR", in2 := 1)
      Coil( "AUTO SUBOUTPUT DB"."PAV-56 INLINE HOMO. SEAL COOLING INLET" )
   END_RUNG
   // the same network as SCL:
   "AUTO SUBOUTPUT DB"."PAV-56 INLINE HOMO. SEAL COOLING INLET" := "AlwaysTRUE" AND ("MODE SELECTION DB"."MODE BUFF" = 1) AND NOT "MFG PROCESS_DB".PAUSE AND ("MFG PROCESS_DB"."AUTO BUFF" = 160) AND ("CONTINUE DB"."SYRUP MFG PROCESS ERROR" <> 1);
END_REGION

REGION Network 49: PBV-57 VACUUM INLET VALVE
   RUNG wire#powerrail
      Contact( "AlwaysTRUE" )
      { S7_Templates := "SrcType := Int" } EQ_Contact(in1 := "MODE SELECTION DB"."MODE BUFF", in2 := 1)
      { S7_Templates := "SrcType := Int" } EQ_Contact(in1 := "MFG PROCESS_DB"."MATERIAL SUCTION"."MATERIAL SUCTION BUFF", in2 := 5)
      { S7_Templates := "SrcType := Int" } NE_Contact(in1 := "LEVEL BUFF".AUTO."MFG VACUUM MIN_MAX BUFF", in2 := 1)
      { S7_Templates := "SrcType := Int" } NE_Contact(in1 := "CONTINUE DB"."SYRUP MFG PROCESS ERROR", in2 := 1)
      Coil( "AUTO SUBOUTPUT DB"."PBV-57 VACUUM INLET VALVE" )
   END_RUNG
   // the same network as SCL:
   "AUTO SUBOUTPUT DB"."PBV-57 VACUUM INLET VALVE" := "AlwaysTRUE" AND ("MODE SELECTION DB"."MODE BUFF" = 1) AND ("MFG PROCESS_DB"."MATERIAL SUCTION"."MATERIAL SUCTION BUFF" = 5) AND ("LEVEL BUFF".AUTO."MFG VACUUM MIN_MAX BUFF" <> 1) AND ("CONTINUE DB"."SYRUP MFG PROCESS ERROR" <> 1);
END_REGION

REGION Network 50: PFBV-59 TANK OUTLET VALVE
   RUNG wire#powerrail
      Contact( "AlwaysTRUE" )
      { S7_Templates := "SrcType := Int" } EQ_Contact(in1 := "MODE SELECTION DB"."MODE BUFF", in2 := 1)
      I_Contact( "MFG PROCESS_DB".PAUSE )
      { S7_Templates := "SrcType := Int" } EQ_Contact(in1 := "MFG PROCESS_DB"."AUTO BUFF", in2 := 160)
      { S7_Templates := "SrcType := Int" } NE_Contact(in1 := "CONTINUE DB"."SYRUP MFG PROCESS ERROR", in2 := 1)
      Coil( "AUTO SUBOUTPUT DB"."PFBV-59 TANK OUTLET VALVE" )
   END_RUNG
   // the same network as SCL:
   "AUTO SUBOUTPUT DB"."PFBV-59 TANK OUTLET VALVE" := "AlwaysTRUE" AND ("MODE SELECTION DB"."MODE BUFF" = 1) AND NOT "MFG PROCESS_DB".PAUSE AND ("MFG PROCESS_DB"."AUTO BUFF" = 160) AND ("CONTINUE DB"."SYRUP MFG PROCESS ERROR" <> 1);
END_REGION

REGION Network 51: PBV-79 BASKET FILTER INLET
   RUNG wire#powerrail
      Contact( "AlwaysFALSE" )
      { S7_Templates := "SrcType := Int" } EQ_Contact(in1 := "MODE SELECTION DB"."MODE BUFF", in2 := 1)
      Coil( "AUTO SUBOUTPUT DB"."PBV-79 BASKET FILTER INLET" )
   END_RUNG
   // the same network as SCL:
   "AUTO SUBOUTPUT DB"."PBV-79 BASKET FILTER INLET" := "AlwaysFALSE" AND ("MODE SELECTION DB"."MODE BUFF" = 1);
END_REGION

REGION Network 52: PBV-80 BOTTOM OUTLET TO BASKET FILTER
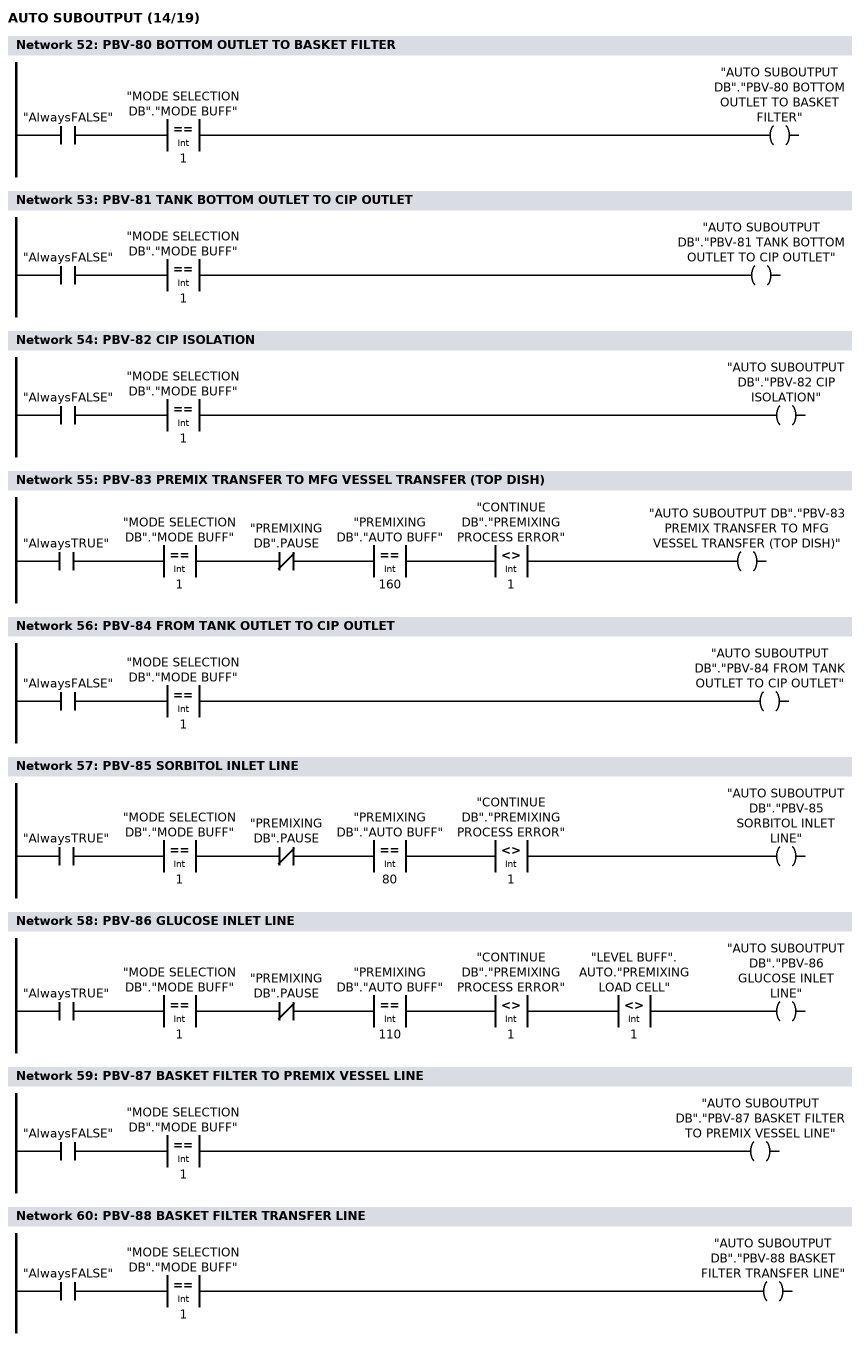
   RUNG wire#powerrail
      Contact( "AlwaysFALSE" )
      { S7_Templates := "SrcType := Int" } EQ_Contact(in1 := "MODE SELECTION DB"."MODE BUFF", in2 := 1)
      Coil( "AUTO SUBOUTPUT DB"."PBV-80 BOTTOM OUTLET TO BASKET FILTER" )
   END_RUNG
   // the same network as SCL:
   "AUTO SUBOUTPUT DB"."PBV-80 BOTTOM OUTLET TO BASKET FILTER" := "AlwaysFALSE" AND ("MODE SELECTION DB"."MODE BUFF" = 1);
END_REGION

REGION Network 53: PBV-81 TANK BOTTOM OUTLET TO CIP OUTLET
   RUNG wire#powerrail
      Contact( "AlwaysFALSE" )
      { S7_Templates := "SrcType := Int" } EQ_Contact(in1 := "MODE SELECTION DB"."MODE BUFF", in2 := 1)
      Coil( "AUTO SUBOUTPUT DB"."PBV-81 TANK BOTTOM OUTLET TO CIP OUTLET" )
   END_RUNG
   // the same network as SCL:
   "AUTO SUBOUTPUT DB"."PBV-81 TANK BOTTOM OUTLET TO CIP OUTLET" := "AlwaysFALSE" AND ("MODE SELECTION DB"."MODE BUFF" = 1);
END_REGION

REGION Network 54: PBV-82 CIP ISOLATION
   RUNG wire#powerrail
      Contact( "AlwaysFALSE" )
      { S7_Templates := "SrcType := Int" } EQ_Contact(in1 := "MODE SELECTION DB"."MODE BUFF", in2 := 1)
      Coil( "AUTO SUBOUTPUT DB"."PBV-82 CIP ISOLATION" )
   END_RUNG
   // the same network as SCL:
   "AUTO SUBOUTPUT DB"."PBV-82 CIP ISOLATION" := "AlwaysFALSE" AND ("MODE SELECTION DB"."MODE BUFF" = 1);
END_REGION

REGION Network 55: PBV-83 PREMIX TRANSFER TO MFG VESSEL TRANSFER (TOP DISH)
   RUNG wire#powerrail
      Contact( "AlwaysTRUE" )
      { S7_Templates := "SrcType := Int" } EQ_Contact(in1 := "MODE SELECTION DB"."MODE BUFF", in2 := 1)
      I_Contact( "PREMIXING DB".PAUSE )
      { S7_Templates := "SrcType := Int" } EQ_Contact(in1 := "PREMIXING DB"."AUTO BUFF", in2 := 160)
      { S7_Templates := "SrcType := Int" } NE_Contact(in1 := "CONTINUE DB"."PREMIXING PROCESS ERROR", in2 := 1)
      Coil( "AUTO SUBOUTPUT DB"."PBV-83 PREMIX TRANSFER TO MFG VESSEL TRANSFER (TOP DISH)" )
   END_RUNG
   // the same network as SCL:
   "AUTO SUBOUTPUT DB"."PBV-83 PREMIX TRANSFER TO MFG VESSEL TRANSFER (TOP DISH)" := "AlwaysTRUE" AND ("MODE SELECTION DB"."MODE BUFF" = 1) AND NOT "PREMIXING DB".PAUSE AND ("PREMIXING DB"."AUTO BUFF" = 160) AND ("CONTINUE DB"."PREMIXING PROCESS ERROR" <> 1);
END_REGION

REGION Network 56: PBV-84 FROM TANK OUTLET TO CIP OUTLET
   RUNG wire#powerrail
      Contact( "AlwaysFALSE" )
      { S7_Templates := "SrcType := Int" } EQ_Contact(in1 := "MODE SELECTION DB"."MODE BUFF", in2 := 1)
      Coil( "AUTO SUBOUTPUT DB"."PBV-84 FROM TANK OUTLET TO CIP OUTLET" )
   END_RUNG
   // the same network as SCL:
   "AUTO SUBOUTPUT DB"."PBV-84 FROM TANK OUTLET TO CIP OUTLET" := "AlwaysFALSE" AND ("MODE SELECTION DB"."MODE BUFF" = 1);
END_REGION

REGION Network 57: PBV-85 SORBITOL INLET LINE
   RUNG wire#powerrail
      Contact( "AlwaysTRUE" )
      { S7_Templates := "SrcType := Int" } EQ_Contact(in1 := "MODE SELECTION DB"."MODE BUFF", in2 := 1)
      I_Contact( "PREMIXING DB".PAUSE )
      { S7_Templates := "SrcType := Int" } EQ_Contact(in1 := "PREMIXING DB"."AUTO BUFF", in2 := 80)
      { S7_Templates := "SrcType := Int" } NE_Contact(in1 := "CONTINUE DB"."PREMIXING PROCESS ERROR", in2 := 1)
      Coil( "AUTO SUBOUTPUT DB"."PBV-85 SORBITOL INLET LINE" )
   END_RUNG
   // the same network as SCL:
   "AUTO SUBOUTPUT DB"."PBV-85 SORBITOL INLET LINE" := "AlwaysTRUE" AND ("MODE SELECTION DB"."MODE BUFF" = 1) AND NOT "PREMIXING DB".PAUSE AND ("PREMIXING DB"."AUTO BUFF" = 80) AND ("CONTINUE DB"."PREMIXING PROCESS ERROR" <> 1);
END_REGION

REGION Network 58: PBV-86 GLUCOSE INLET LINE
   RUNG wire#powerrail
      Contact( "AlwaysTRUE" )
      { S7_Templates := "SrcType := Int" } EQ_Contact(in1 := "MODE SELECTION DB"."MODE BUFF", in2 := 1)
      I_Contact( "PREMIXING DB".PAUSE )
      { S7_Templates := "SrcType := Int" } EQ_Contact(in1 := "PREMIXING DB"."AUTO BUFF", in2 := 110)
      { S7_Templates := "SrcType := Int" } NE_Contact(in1 := "CONTINUE DB"."PREMIXING PROCESS ERROR", in2 := 1)
      { S7_Templates := "SrcType := Int" } NE_Contact(in1 := "LEVEL BUFF".AUTO."PREMIXING LOAD CELL", in2 := 1)
      Coil( "AUTO SUBOUTPUT DB"."PBV-86 GLUCOSE INLET LINE" )
   END_RUNG
   // the same network as SCL:
   "AUTO SUBOUTPUT DB"."PBV-86 GLUCOSE INLET LINE" := "AlwaysTRUE" AND ("MODE SELECTION DB"."MODE BUFF" = 1) AND NOT "PREMIXING DB".PAUSE AND ("PREMIXING DB"."AUTO BUFF" = 110) AND ("CONTINUE DB"."PREMIXING PROCESS ERROR" <> 1) AND ("LEVEL BUFF".AUTO."PREMIXING LOAD CELL" <> 1);
END_REGION

REGION Network 59: PBV-87 BASKET FILTER TO PREMIX VESSEL LINE
   RUNG wire#powerrail
      Contact( "AlwaysFALSE" )
      { S7_Templates := "SrcType := Int" } EQ_Contact(in1 := "MODE SELECTION DB"."MODE BUFF", in2 := 1)
      Coil( "AUTO SUBOUTPUT DB"."PBV-87 BASKET FILTER TO PREMIX VESSEL LINE" )
   END_RUNG
   // the same network as SCL:
   "AUTO SUBOUTPUT DB"."PBV-87 BASKET FILTER TO PREMIX VESSEL LINE" := "AlwaysFALSE" AND ("MODE SELECTION DB"."MODE BUFF" = 1);
END_REGION

REGION Network 60: PBV-88 BASKET FILTER TRANSFER LINE
   RUNG wire#powerrail
      Contact( "AlwaysFALSE" )
      { S7_Templates := "SrcType := Int" } EQ_Contact(in1 := "MODE SELECTION DB"."MODE BUFF", in2 := 1)
      Coil( "AUTO SUBOUTPUT DB"."PBV-88 BASKET FILTER TRANSFER LINE" )
   END_RUNG
   // the same network as SCL:
   "AUTO SUBOUTPUT DB"."PBV-88 BASKET FILTER TRANSFER LINE" := "AlwaysFALSE" AND ("MODE SELECTION DB"."MODE BUFF" = 1);
END_REGION

REGION Network 61: PBV-89 BASKET FILTER TO MFG INLET TRANSFER LINE
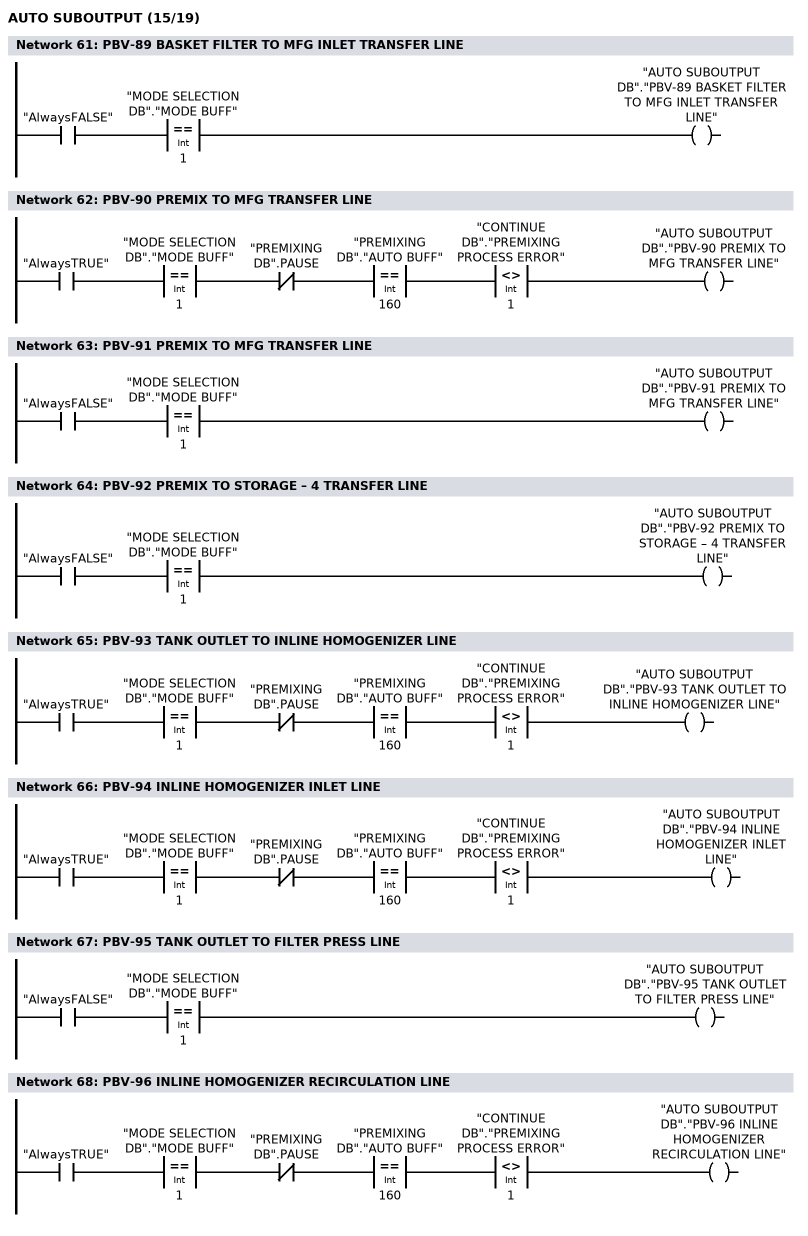
   RUNG wire#powerrail
      Contact( "AlwaysFALSE" )
      { S7_Templates := "SrcType := Int" } EQ_Contact(in1 := "MODE SELECTION DB"."MODE BUFF", in2 := 1)
      Coil( "AUTO SUBOUTPUT DB"."PBV-89 BASKET FILTER TO MFG INLET TRANSFER LINE" )
   END_RUNG
   // the same network as SCL:
   "AUTO SUBOUTPUT DB"."PBV-89 BASKET FILTER TO MFG INLET TRANSFER LINE" := "AlwaysFALSE" AND ("MODE SELECTION DB"."MODE BUFF" = 1);
END_REGION

REGION Network 62: PBV-90 PREMIX TO MFG TRANSFER LINE
   RUNG wire#powerrail
      Contact( "AlwaysTRUE" )
      { S7_Templates := "SrcType := Int" } EQ_Contact(in1 := "MODE SELECTION DB"."MODE BUFF", in2 := 1)
      I_Contact( "PREMIXING DB".PAUSE )
      { S7_Templates := "SrcType := Int" } EQ_Contact(in1 := "PREMIXING DB"."AUTO BUFF", in2 := 160)
      { S7_Templates := "SrcType := Int" } NE_Contact(in1 := "CONTINUE DB"."PREMIXING PROCESS ERROR", in2 := 1)
      Coil( "AUTO SUBOUTPUT DB"."PBV-90 PREMIX TO MFG TRANSFER LINE" )
   END_RUNG
   // the same network as SCL:
   "AUTO SUBOUTPUT DB"."PBV-90 PREMIX TO MFG TRANSFER LINE" := "AlwaysTRUE" AND ("MODE SELECTION DB"."MODE BUFF" = 1) AND NOT "PREMIXING DB".PAUSE AND ("PREMIXING DB"."AUTO BUFF" = 160) AND ("CONTINUE DB"."PREMIXING PROCESS ERROR" <> 1);
END_REGION

REGION Network 63: PBV-91 PREMIX TO MFG TRANSFER LINE
   RUNG wire#powerrail
      Contact( "AlwaysFALSE" )
      { S7_Templates := "SrcType := Int" } EQ_Contact(in1 := "MODE SELECTION DB"."MODE BUFF", in2 := 1)
      Coil( "AUTO SUBOUTPUT DB"."PBV-91 PREMIX TO MFG TRANSFER LINE" )
   END_RUNG
   // the same network as SCL:
   "AUTO SUBOUTPUT DB"."PBV-91 PREMIX TO MFG TRANSFER LINE" := "AlwaysFALSE" AND ("MODE SELECTION DB"."MODE BUFF" = 1);
END_REGION

REGION Network 64: PBV-92 PREMIX TO STORAGE – 4 TRANSFER LINE
   RUNG wire#powerrail
      Contact( "AlwaysFALSE" )
      { S7_Templates := "SrcType := Int" } EQ_Contact(in1 := "MODE SELECTION DB"."MODE BUFF", in2 := 1)
      Coil( "AUTO SUBOUTPUT DB"."PBV-92 PREMIX TO STORAGE – 4 TRANSFER LINE" )
   END_RUNG
   // the same network as SCL:
   "AUTO SUBOUTPUT DB"."PBV-92 PREMIX TO STORAGE – 4 TRANSFER LINE" := "AlwaysFALSE" AND ("MODE SELECTION DB"."MODE BUFF" = 1);
END_REGION

REGION Network 65: PBV-93 TANK OUTLET TO INLINE HOMOGENIZER LINE
   RUNG wire#powerrail
      Contact( "AlwaysTRUE" )
      { S7_Templates := "SrcType := Int" } EQ_Contact(in1 := "MODE SELECTION DB"."MODE BUFF", in2 := 1)
      I_Contact( "PREMIXING DB".PAUSE )
      { S7_Templates := "SrcType := Int" } EQ_Contact(in1 := "PREMIXING DB"."AUTO BUFF", in2 := 160)
      { S7_Templates := "SrcType := Int" } NE_Contact(in1 := "CONTINUE DB"."PREMIXING PROCESS ERROR", in2 := 1)
      Coil( "AUTO SUBOUTPUT DB"."PBV-93 TANK OUTLET TO INLINE HOMOGENIZER LINE" )
   END_RUNG
   // the same network as SCL:
   "AUTO SUBOUTPUT DB"."PBV-93 TANK OUTLET TO INLINE HOMOGENIZER LINE" := "AlwaysTRUE" AND ("MODE SELECTION DB"."MODE BUFF" = 1) AND NOT "PREMIXING DB".PAUSE AND ("PREMIXING DB"."AUTO BUFF" = 160) AND ("CONTINUE DB"."PREMIXING PROCESS ERROR" <> 1);
END_REGION

REGION Network 66: PBV-94 INLINE HOMOGENIZER INLET LINE
   RUNG wire#powerrail
      Contact( "AlwaysTRUE" )
      { S7_Templates := "SrcType := Int" } EQ_Contact(in1 := "MODE SELECTION DB"."MODE BUFF", in2 := 1)
      I_Contact( "PREMIXING DB".PAUSE )
      { S7_Templates := "SrcType := Int" } EQ_Contact(in1 := "PREMIXING DB"."AUTO BUFF", in2 := 160)
      { S7_Templates := "SrcType := Int" } NE_Contact(in1 := "CONTINUE DB"."PREMIXING PROCESS ERROR", in2 := 1)
      Coil( "AUTO SUBOUTPUT DB"."PBV-94 INLINE HOMOGENIZER INLET LINE" )
   END_RUNG
   // the same network as SCL:
   "AUTO SUBOUTPUT DB"."PBV-94 INLINE HOMOGENIZER INLET LINE" := "AlwaysTRUE" AND ("MODE SELECTION DB"."MODE BUFF" = 1) AND NOT "PREMIXING DB".PAUSE AND ("PREMIXING DB"."AUTO BUFF" = 160) AND ("CONTINUE DB"."PREMIXING PROCESS ERROR" <> 1);
END_REGION

REGION Network 67: PBV-95 TANK OUTLET TO FILTER PRESS LINE
   RUNG wire#powerrail
      Contact( "AlwaysFALSE" )
      { S7_Templates := "SrcType := Int" } EQ_Contact(in1 := "MODE SELECTION DB"."MODE BUFF", in2 := 1)
      Coil( "AUTO SUBOUTPUT DB"."PBV-95 TANK OUTLET TO FILTER PRESS LINE" )
   END_RUNG
   // the same network as SCL:
   "AUTO SUBOUTPUT DB"."PBV-95 TANK OUTLET TO FILTER PRESS LINE" := "AlwaysFALSE" AND ("MODE SELECTION DB"."MODE BUFF" = 1);
END_REGION

REGION Network 68: PBV-96 INLINE HOMOGENIZER RECIRCULATION LINE
   RUNG wire#powerrail
      Contact( "AlwaysTRUE" )
      { S7_Templates := "SrcType := Int" } EQ_Contact(in1 := "MODE SELECTION DB"."MODE BUFF", in2 := 1)
      I_Contact( "PREMIXING DB".PAUSE )
      { S7_Templates := "SrcType := Int" } EQ_Contact(in1 := "PREMIXING DB"."AUTO BUFF", in2 := 160)
      { S7_Templates := "SrcType := Int" } NE_Contact(in1 := "CONTINUE DB"."PREMIXING PROCESS ERROR", in2 := 1)
      Coil( "AUTO SUBOUTPUT DB"."PBV-96 INLINE HOMOGENIZER RECIRCULATION LINE" )
   END_RUNG
   // the same network as SCL:
   "AUTO SUBOUTPUT DB"."PBV-96 INLINE HOMOGENIZER RECIRCULATION LINE" := "AlwaysTRUE" AND ("MODE SELECTION DB"."MODE BUFF" = 1) AND NOT "PREMIXING DB".PAUSE AND ("PREMIXING DB"."AUTO BUFF" = 160) AND ("CONTINUE DB"."PREMIXING PROCESS ERROR" <> 1);
END_REGION

REGION Network 69: PBV-97 FILTER PRESS OUTLET
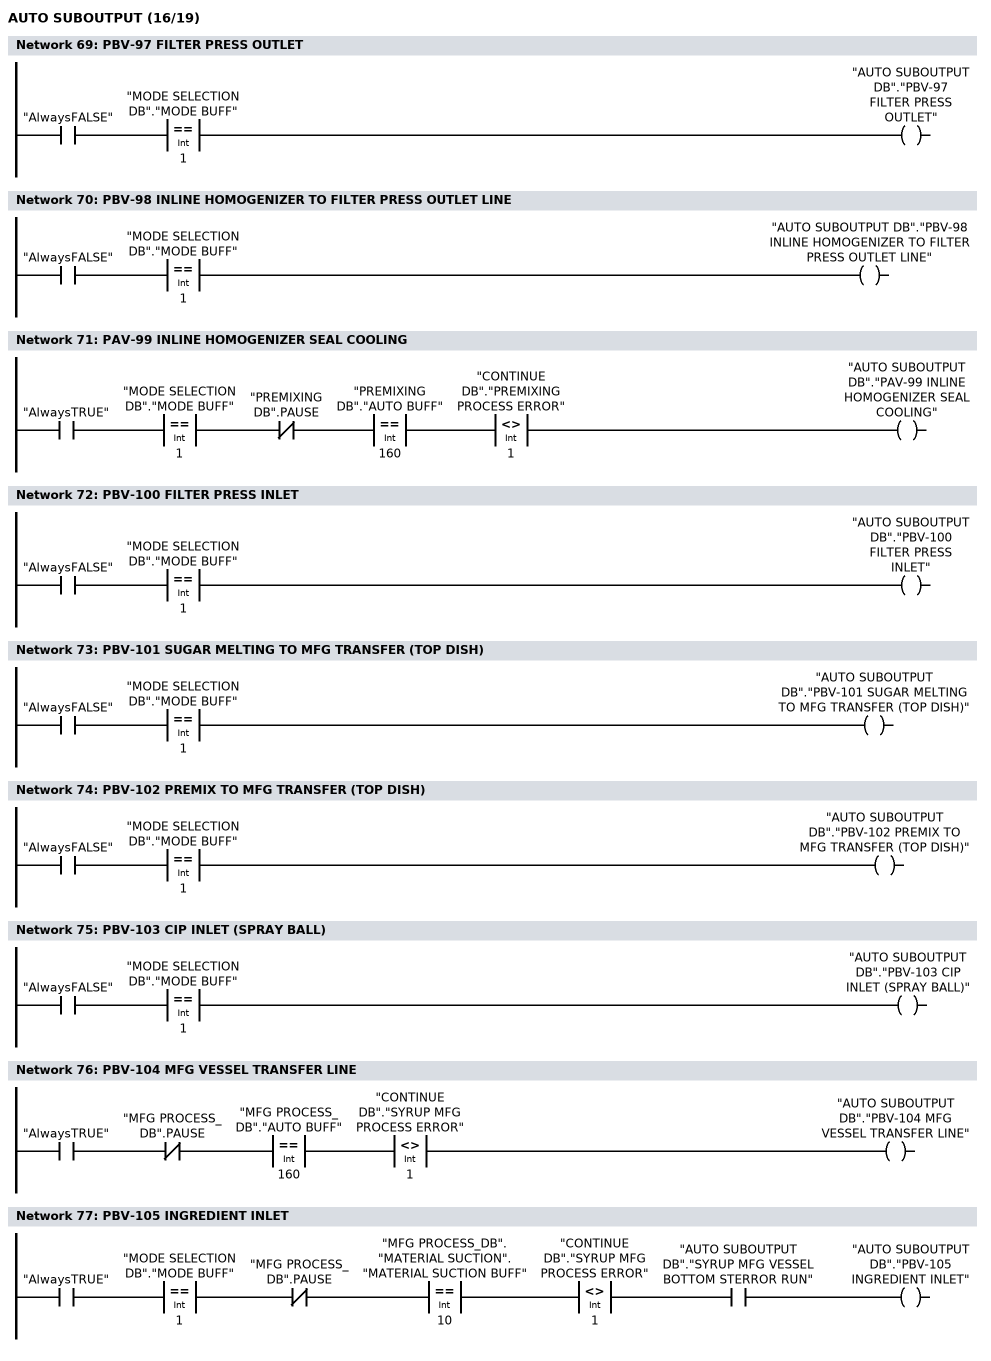
   RUNG wire#powerrail
      Contact( "AlwaysFALSE" )
      { S7_Templates := "SrcType := Int" } EQ_Contact(in1 := "MODE SELECTION DB"."MODE BUFF", in2 := 1)
      Coil( "AUTO SUBOUTPUT DB"."PBV-97 FILTER PRESS OUTLET" )
   END_RUNG
   // the same network as SCL:
   "AUTO SUBOUTPUT DB"."PBV-97 FILTER PRESS OUTLET" := "AlwaysFALSE" AND ("MODE SELECTION DB"."MODE BUFF" = 1);
END_REGION

REGION Network 70: PBV-98 INLINE HOMOGENIZER TO FILTER PRESS OUTLET LINE
   RUNG wire#powerrail
      Contact( "AlwaysFALSE" )
      { S7_Templates := "SrcType := Int" } EQ_Contact(in1 := "MODE SELECTION DB"."MODE BUFF", in2 := 1)
      Coil( "AUTO SUBOUTPUT DB"."PBV-98 INLINE HOMOGENIZER TO FILTER PRESS OUTLET LINE" )
   END_RUNG
   // the same network as SCL:
   "AUTO SUBOUTPUT DB"."PBV-98 INLINE HOMOGENIZER TO FILTER PRESS OUTLET LINE" := "AlwaysFALSE" AND ("MODE SELECTION DB"."MODE BUFF" = 1);
END_REGION

REGION Network 71: PAV-99 INLINE HOMOGENIZER SEAL COOLING
   RUNG wire#powerrail
      Contact( "AlwaysTRUE" )
      { S7_Templates := "SrcType := Int" } EQ_Contact(in1 := "MODE SELECTION DB"."MODE BUFF", in2 := 1)
      I_Contact( "PREMIXING DB".PAUSE )
      { S7_Templates := "SrcType := Int" } EQ_Contact(in1 := "PREMIXING DB"."AUTO BUFF", in2 := 160)
      { S7_Templates := "SrcType := Int" } NE_Contact(in1 := "CONTINUE DB"."PREMIXING PROCESS ERROR", in2 := 1)
      Coil( "AUTO SUBOUTPUT DB"."PAV-99 INLINE HOMOGENIZER SEAL COOLING" )
   END_RUNG
   // the same network as SCL:
   "AUTO SUBOUTPUT DB"."PAV-99 INLINE HOMOGENIZER SEAL COOLING" := "AlwaysTRUE" AND ("MODE SELECTION DB"."MODE BUFF" = 1) AND NOT "PREMIXING DB".PAUSE AND ("PREMIXING DB"."AUTO BUFF" = 160) AND ("CONTINUE DB"."PREMIXING PROCESS ERROR" <> 1);
END_REGION

REGION Network 72: PBV-100 FILTER PRESS INLET
   RUNG wire#powerrail
      Contact( "AlwaysFALSE" )
      { S7_Templates := "SrcType := Int" } EQ_Contact(in1 := "MODE SELECTION DB"."MODE BUFF", in2 := 1)
      Coil( "AUTO SUBOUTPUT DB"."PBV-100 FILTER PRESS INLET" )
   END_RUNG
   // the same network as SCL:
   "AUTO SUBOUTPUT DB"."PBV-100 FILTER PRESS INLET" := "AlwaysFALSE" AND ("MODE SELECTION DB"."MODE BUFF" = 1);
END_REGION

REGION Network 73: PBV-101 SUGAR MELTING TO MFG TRANSFER (TOP DISH)
   RUNG wire#powerrail
      Contact( "AlwaysFALSE" )
      { S7_Templates := "SrcType := Int" } EQ_Contact(in1 := "MODE SELECTION DB"."MODE BUFF", in2 := 1)
      Coil( "AUTO SUBOUTPUT DB"."PBV-101 SUGAR MELTING TO MFG TRANSFER (TOP DISH)" )
   END_RUNG
   // the same network as SCL:
   "AUTO SUBOUTPUT DB"."PBV-101 SUGAR MELTING TO MFG TRANSFER (TOP DISH)" := "AlwaysFALSE" AND ("MODE SELECTION DB"."MODE BUFF" = 1);
END_REGION

REGION Network 74: PBV-102 PREMIX TO MFG TRANSFER (TOP DISH)
   RUNG wire#powerrail
      Contact( "AlwaysFALSE" )
      { S7_Templates := "SrcType := Int" } EQ_Contact(in1 := "MODE SELECTION DB"."MODE BUFF", in2 := 1)
      Coil( "AUTO SUBOUTPUT DB"."PBV-102 PREMIX TO MFG TRANSFER (TOP DISH)" )
   END_RUNG
   // the same network as SCL:
   "AUTO SUBOUTPUT DB"."PBV-102 PREMIX TO MFG TRANSFER (TOP DISH)" := "AlwaysFALSE" AND ("MODE SELECTION DB"."MODE BUFF" = 1);
END_REGION

REGION Network 75: PBV-103 CIP INLET (SPRAY BALL)
   RUNG wire#powerrail
      Contact( "AlwaysFALSE" )
      { S7_Templates := "SrcType := Int" } EQ_Contact(in1 := "MODE SELECTION DB"."MODE BUFF", in2 := 1)
      Coil( "AUTO SUBOUTPUT DB"."PBV-103 CIP INLET (SPRAY BALL)" )
   END_RUNG
   // the same network as SCL:
   "AUTO SUBOUTPUT DB"."PBV-103 CIP INLET (SPRAY BALL)" := "AlwaysFALSE" AND ("MODE SELECTION DB"."MODE BUFF" = 1);
END_REGION

REGION Network 76: PBV-104 MFG VESSEL TRANSFER LINE
   RUNG wire#powerrail
      Contact( "AlwaysTRUE" )
      I_Contact( "MFG PROCESS_DB".PAUSE )
      { S7_Templates := "SrcType := Int" } EQ_Contact(in1 := "MFG PROCESS_DB"."AUTO BUFF", in2 := 160)
      { S7_Templates := "SrcType := Int" } NE_Contact(in1 := "CONTINUE DB"."SYRUP MFG PROCESS ERROR", in2 := 1)
      Coil( "AUTO SUBOUTPUT DB"."PBV-104 MFG VESSEL TRANSFER LINE" )
   END_RUNG
   // the same network as SCL:
   "AUTO SUBOUTPUT DB"."PBV-104 MFG VESSEL TRANSFER LINE" := "AlwaysTRUE" AND NOT "MFG PROCESS_DB".PAUSE AND ("MFG PROCESS_DB"."AUTO BUFF" = 160) AND ("CONTINUE DB"."SYRUP MFG PROCESS ERROR" <> 1);
END_REGION

REGION Network 77: PBV-105 INGREDIENT INLET
   RUNG wire#powerrail
      Contact( "AlwaysTRUE" )
      { S7_Templates := "SrcType := Int" } EQ_Contact(in1 := "MODE SELECTION DB"."MODE BUFF", in2 := 1)
      I_Contact( "MFG PROCESS_DB".PAUSE )
      { S7_Templates := "SrcType := Int" } EQ_Contact(in1 := "MFG PROCESS_DB"."MATERIAL SUCTION"."MATERIAL SUCTION BUFF", in2 := 10)
      { S7_Templates := "SrcType := Int" } NE_Contact(in1 := "CONTINUE DB"."SYRUP MFG PROCESS ERROR", in2 := 1)
      Contact( "AUTO SUBOUTPUT DB"."SYRUP MFG VESSEL BOTTOM STERROR RUN" )
      Coil( "AUTO SUBOUTPUT DB"."PBV-105 INGREDIENT INLET" )
   END_RUNG
   // the same network as SCL:
   "AUTO SUBOUTPUT DB"."PBV-105 INGREDIENT INLET" := "AlwaysTRUE" AND ("MODE SELECTION DB"."MODE BUFF" = 1) AND NOT "MFG PROCESS_DB".PAUSE AND ("MFG PROCESS_DB"."MATERIAL SUCTION"."MATERIAL SUCTION BUFF" = 10) AND ("CONTINUE DB"."SYRUP MFG PROCESS ERROR" <> 1) AND "AUTO SUBOUTPUT DB"."SYRUP MFG VESSEL BOTTOM STERROR RUN";
END_REGION

REGION Network 78: PBV-106 SORBITOL INLET
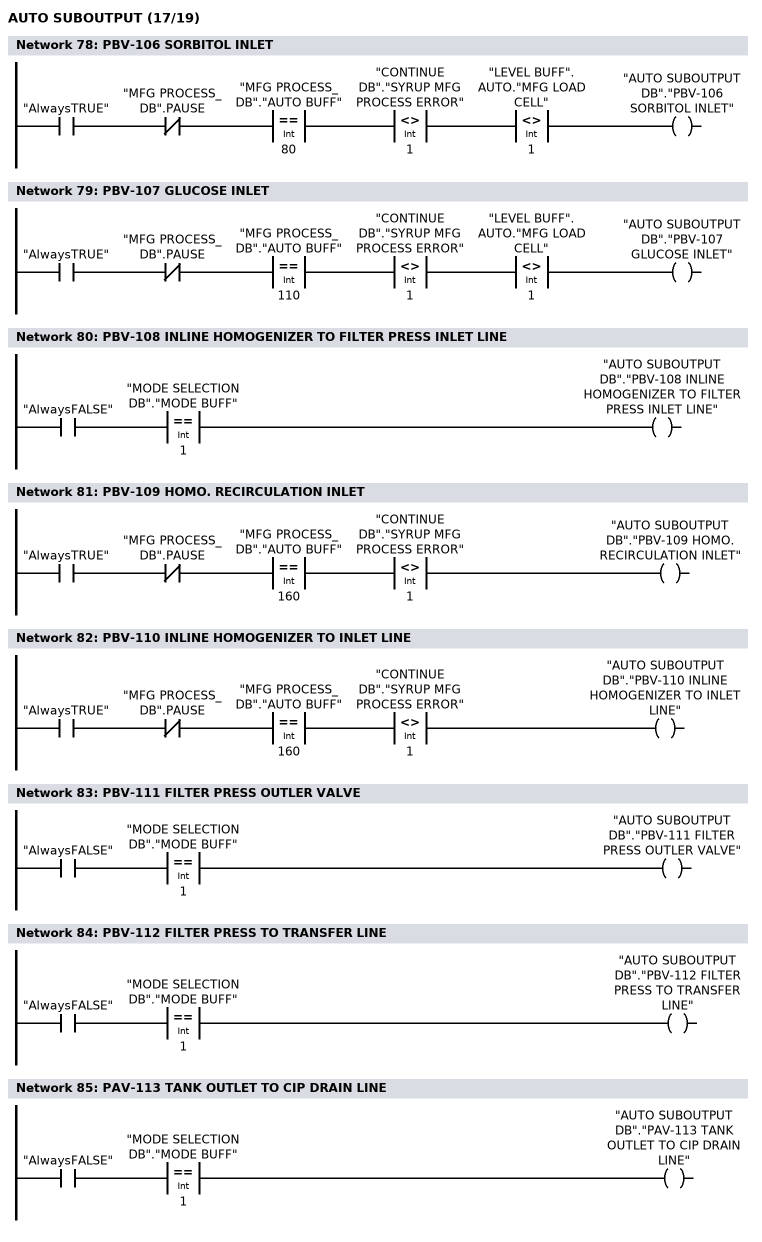
   RUNG wire#powerrail
      Contact( "AlwaysTRUE" )
      I_Contact( "MFG PROCESS_DB".PAUSE )
      { S7_Templates := "SrcType := Int" } EQ_Contact(in1 := "MFG PROCESS_DB"."AUTO BUFF", in2 := 80)
      { S7_Templates := "SrcType := Int" } NE_Contact(in1 := "CONTINUE DB"."SYRUP MFG PROCESS ERROR", in2 := 1)
      { S7_Templates := "SrcType := Int" } NE_Contact(in1 := "LEVEL BUFF".AUTO."MFG LOAD CELL", in2 := 1)
      Coil( "AUTO SUBOUTPUT DB"."PBV-106 SORBITOL INLET" )
   END_RUNG
   // the same network as SCL:
   "AUTO SUBOUTPUT DB"."PBV-106 SORBITOL INLET" := "AlwaysTRUE" AND NOT "MFG PROCESS_DB".PAUSE AND ("MFG PROCESS_DB"."AUTO BUFF" = 80) AND ("CONTINUE DB"."SYRUP MFG PROCESS ERROR" <> 1) AND ("LEVEL BUFF".AUTO."MFG LOAD CELL" <> 1);
END_REGION

REGION Network 79: PBV-107 GLUCOSE INLET
   RUNG wire#powerrail
      Contact( "AlwaysTRUE" )
      I_Contact( "MFG PROCESS_DB".PAUSE )
      { S7_Templates := "SrcType := Int" } EQ_Contact(in1 := "MFG PROCESS_DB"."AUTO BUFF", in2 := 110)
      { S7_Templates := "SrcType := Int" } NE_Contact(in1 := "CONTINUE DB"."SYRUP MFG PROCESS ERROR", in2 := 1)
      { S7_Templates := "SrcType := Int" } NE_Contact(in1 := "LEVEL BUFF".AUTO."MFG LOAD CELL", in2 := 1)
      Coil( "AUTO SUBOUTPUT DB"."PBV-107 GLUCOSE INLET" )
   END_RUNG
   // the same network as SCL:
   "AUTO SUBOUTPUT DB"."PBV-107 GLUCOSE INLET" := "AlwaysTRUE" AND NOT "MFG PROCESS_DB".PAUSE AND ("MFG PROCESS_DB"."AUTO BUFF" = 110) AND ("CONTINUE DB"."SYRUP MFG PROCESS ERROR" <> 1) AND ("LEVEL BUFF".AUTO."MFG LOAD CELL" <> 1);
END_REGION

REGION Network 80: PBV-108 INLINE HOMOGENIZER TO FILTER PRESS INLET LINE
   RUNG wire#powerrail
      Contact( "AlwaysFALSE" )
      { S7_Templates := "SrcType := Int" } EQ_Contact(in1 := "MODE SELECTION DB"."MODE BUFF", in2 := 1)
      Coil( "AUTO SUBOUTPUT DB"."PBV-108 INLINE HOMOGENIZER TO FILTER PRESS INLET LINE" )
   END_RUNG
   // the same network as SCL:
   "AUTO SUBOUTPUT DB"."PBV-108 INLINE HOMOGENIZER TO FILTER PRESS INLET LINE" := "AlwaysFALSE" AND ("MODE SELECTION DB"."MODE BUFF" = 1);
END_REGION

REGION Network 81: PBV-109 HOMO. RECIRCULATION INLET
   RUNG wire#powerrail
      Contact( "AlwaysTRUE" )
      I_Contact( "MFG PROCESS_DB".PAUSE )
      { S7_Templates := "SrcType := Int" } EQ_Contact(in1 := "MFG PROCESS_DB"."AUTO BUFF", in2 := 160)
      { S7_Templates := "SrcType := Int" } NE_Contact(in1 := "CONTINUE DB"."SYRUP MFG PROCESS ERROR", in2 := 1)
      Coil( "AUTO SUBOUTPUT DB"."PBV-109 HOMO. RECIRCULATION INLET" )
   END_RUNG
   // the same network as SCL:
   "AUTO SUBOUTPUT DB"."PBV-109 HOMO. RECIRCULATION INLET" := "AlwaysTRUE" AND NOT "MFG PROCESS_DB".PAUSE AND ("MFG PROCESS_DB"."AUTO BUFF" = 160) AND ("CONTINUE DB"."SYRUP MFG PROCESS ERROR" <> 1);
END_REGION

REGION Network 82: PBV-110 INLINE HOMOGENIZER TO INLET LINE
   RUNG wire#powerrail
      Contact( "AlwaysTRUE" )
      I_Contact( "MFG PROCESS_DB".PAUSE )
      { S7_Templates := "SrcType := Int" } EQ_Contact(in1 := "MFG PROCESS_DB"."AUTO BUFF", in2 := 160)
      { S7_Templates := "SrcType := Int" } NE_Contact(in1 := "CONTINUE DB"."SYRUP MFG PROCESS ERROR", in2 := 1)
      Coil( "AUTO SUBOUTPUT DB"."PBV-110 INLINE HOMOGENIZER TO INLET LINE" )
   END_RUNG
   // the same network as SCL:
   "AUTO SUBOUTPUT DB"."PBV-110 INLINE HOMOGENIZER TO INLET LINE" := "AlwaysTRUE" AND NOT "MFG PROCESS_DB".PAUSE AND ("MFG PROCESS_DB"."AUTO BUFF" = 160) AND ("CONTINUE DB"."SYRUP MFG PROCESS ERROR" <> 1);
END_REGION

REGION Network 83: PBV-111 FILTER PRESS OUTLER VALVE
   RUNG wire#powerrail
      Contact( "AlwaysFALSE" )
      { S7_Templates := "SrcType := Int" } EQ_Contact(in1 := "MODE SELECTION DB"."MODE BUFF", in2 := 1)
      Coil( "AUTO SUBOUTPUT DB"."PBV-111 FILTER PRESS OUTLER VALVE" )
   END_RUNG
   // the same network as SCL:
   "AUTO SUBOUTPUT DB"."PBV-111 FILTER PRESS OUTLER VALVE" := "AlwaysFALSE" AND ("MODE SELECTION DB"."MODE BUFF" = 1);
END_REGION

REGION Network 84: PBV-112 FILTER PRESS TO TRANSFER LINE
   RUNG wire#powerrail
      Contact( "AlwaysFALSE" )
      { S7_Templates := "SrcType := Int" } EQ_Contact(in1 := "MODE SELECTION DB"."MODE BUFF", in2 := 1)
      Coil( "AUTO SUBOUTPUT DB"."PBV-112 FILTER PRESS TO TRANSFER LINE" )
   END_RUNG
   // the same network as SCL:
   "AUTO SUBOUTPUT DB"."PBV-112 FILTER PRESS TO TRANSFER LINE" := "AlwaysFALSE" AND ("MODE SELECTION DB"."MODE BUFF" = 1);
END_REGION

REGION Network 85: PAV-113 TANK OUTLET TO CIP DRAIN LINE
   RUNG wire#powerrail
      Contact( "AlwaysFALSE" )
      { S7_Templates := "SrcType := Int" } EQ_Contact(in1 := "MODE SELECTION DB"."MODE BUFF", in2 := 1)
      Coil( "AUTO SUBOUTPUT DB"."PAV-113 TANK OUTLET TO CIP DRAIN LINE" )
   END_RUNG
   // the same network as SCL:
   "AUTO SUBOUTPUT DB"."PAV-113 TANK OUTLET TO CIP DRAIN LINE" := "AlwaysFALSE" AND ("MODE SELECTION DB"."MODE BUFF" = 1);
END_REGION

REGION Network 86: PBV-114 TANK OUTLET TO INLINE HOMOGENIZER LINE
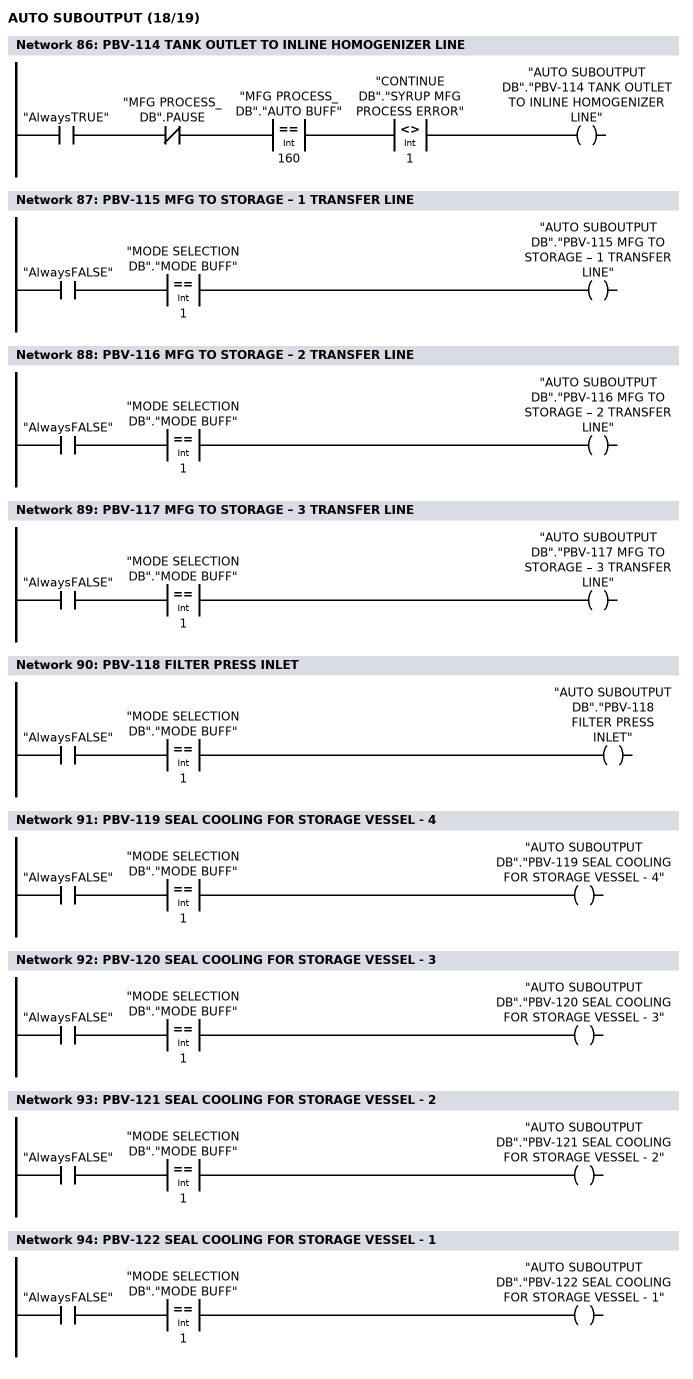
   RUNG wire#powerrail
      Contact( "AlwaysTRUE" )
      I_Contact( "MFG PROCESS_DB".PAUSE )
      { S7_Templates := "SrcType := Int" } EQ_Contact(in1 := "MFG PROCESS_DB"."AUTO BUFF", in2 := 160)
      { S7_Templates := "SrcType := Int" } NE_Contact(in1 := "CONTINUE DB"."SYRUP MFG PROCESS ERROR", in2 := 1)
      Coil( "AUTO SUBOUTPUT DB"."PBV-114 TANK OUTLET TO INLINE HOMOGENIZER LINE" )
   END_RUNG
   // the same network as SCL:
   "AUTO SUBOUTPUT DB"."PBV-114 TANK OUTLET TO INLINE HOMOGENIZER LINE" := "AlwaysTRUE" AND NOT "MFG PROCESS_DB".PAUSE AND ("MFG PROCESS_DB"."AUTO BUFF" = 160) AND ("CONTINUE DB"."SYRUP MFG PROCESS ERROR" <> 1);
END_REGION

REGION Network 87: PBV-115 MFG TO STORAGE – 1 TRANSFER LINE
   RUNG wire#powerrail
      Contact( "AlwaysFALSE" )
      { S7_Templates := "SrcType := Int" } EQ_Contact(in1 := "MODE SELECTION DB"."MODE BUFF", in2 := 1)
      Coil( "AUTO SUBOUTPUT DB"."PBV-115 MFG TO STORAGE – 1 TRANSFER LINE" )
   END_RUNG
   // the same network as SCL:
   "AUTO SUBOUTPUT DB"."PBV-115 MFG TO STORAGE – 1 TRANSFER LINE" := "AlwaysFALSE" AND ("MODE SELECTION DB"."MODE BUFF" = 1);
END_REGION

REGION Network 88: PBV-116 MFG TO STORAGE – 2 TRANSFER LINE
   RUNG wire#powerrail
      Contact( "AlwaysFALSE" )
      { S7_Templates := "SrcType := Int" } EQ_Contact(in1 := "MODE SELECTION DB"."MODE BUFF", in2 := 1)
      Coil( "AUTO SUBOUTPUT DB"."PBV-116 MFG TO STORAGE – 2 TRANSFER LINE" )
   END_RUNG
   // the same network as SCL:
   "AUTO SUBOUTPUT DB"."PBV-116 MFG TO STORAGE – 2 TRANSFER LINE" := "AlwaysFALSE" AND ("MODE SELECTION DB"."MODE BUFF" = 1);
END_REGION

REGION Network 89: PBV-117 MFG TO STORAGE – 3 TRANSFER LINE
   RUNG wire#powerrail
      Contact( "AlwaysFALSE" )
      { S7_Templates := "SrcType := Int" } EQ_Contact(in1 := "MODE SELECTION DB"."MODE BUFF", in2 := 1)
      Coil( "AUTO SUBOUTPUT DB"."PBV-117 MFG TO STORAGE – 3 TRANSFER LINE" )
   END_RUNG
   // the same network as SCL:
   "AUTO SUBOUTPUT DB"."PBV-117 MFG TO STORAGE – 3 TRANSFER LINE" := "AlwaysFALSE" AND ("MODE SELECTION DB"."MODE BUFF" = 1);
END_REGION

REGION Network 90: PBV-118 FILTER PRESS INLET
   RUNG wire#powerrail
      Contact( "AlwaysFALSE" )
      { S7_Templates := "SrcType := Int" } EQ_Contact(in1 := "MODE SELECTION DB"."MODE BUFF", in2 := 1)
      Coil( "AUTO SUBOUTPUT DB"."PBV-118 FILTER PRESS INLET" )
   END_RUNG
   // the same network as SCL:
   "AUTO SUBOUTPUT DB"."PBV-118 FILTER PRESS INLET" := "AlwaysFALSE" AND ("MODE SELECTION DB"."MODE BUFF" = 1);
END_REGION

REGION Network 91: PBV-119 SEAL COOLING FOR STORAGE VESSEL - 4
   RUNG wire#powerrail
      Contact( "AlwaysFALSE" )
      { S7_Templates := "SrcType := Int" } EQ_Contact(in1 := "MODE SELECTION DB"."MODE BUFF", in2 := 1)
      Coil( "AUTO SUBOUTPUT DB"."PBV-119 SEAL COOLING FOR STORAGE VESSEL - 4" )
   END_RUNG
   // the same network as SCL:
   "AUTO SUBOUTPUT DB"."PBV-119 SEAL COOLING FOR STORAGE VESSEL - 4" := "AlwaysFALSE" AND ("MODE SELECTION DB"."MODE BUFF" = 1);
END_REGION

REGION Network 92: PBV-120 SEAL COOLING FOR STORAGE VESSEL - 3
   RUNG wire#powerrail
      Contact( "AlwaysFALSE" )
      { S7_Templates := "SrcType := Int" } EQ_Contact(in1 := "MODE SELECTION DB"."MODE BUFF", in2 := 1)
      Coil( "AUTO SUBOUTPUT DB"."PBV-120 SEAL COOLING FOR STORAGE VESSEL - 3" )
   END_RUNG
   // the same network as SCL:
   "AUTO SUBOUTPUT DB"."PBV-120 SEAL COOLING FOR STORAGE VESSEL - 3" := "AlwaysFALSE" AND ("MODE SELECTION DB"."MODE BUFF" = 1);
END_REGION

REGION Network 93: PBV-121 SEAL COOLING FOR STORAGE VESSEL - 2
   RUNG wire#powerrail
      Contact( "AlwaysFALSE" )
      { S7_Templates := "SrcType := Int" } EQ_Contact(in1 := "MODE SELECTION DB"."MODE BUFF", in2 := 1)
      Coil( "AUTO SUBOUTPUT DB"."PBV-121 SEAL COOLING FOR STORAGE VESSEL - 2" )
   END_RUNG
   // the same network as SCL:
   "AUTO SUBOUTPUT DB"."PBV-121 SEAL COOLING FOR STORAGE VESSEL - 2" := "AlwaysFALSE" AND ("MODE SELECTION DB"."MODE BUFF" = 1);
END_REGION

REGION Network 94: PBV-122 SEAL COOLING FOR STORAGE VESSEL - 1
   RUNG wire#powerrail
      Contact( "AlwaysFALSE" )
      { S7_Templates := "SrcType := Int" } EQ_Contact(in1 := "MODE SELECTION DB"."MODE BUFF", in2 := 1)
      Coil( "AUTO SUBOUTPUT DB"."PBV-122 SEAL COOLING FOR STORAGE VESSEL - 1" )
   END_RUNG
   // the same network as SCL:
   "AUTO SUBOUTPUT DB"."PBV-122 SEAL COOLING FOR STORAGE VESSEL - 1" := "AlwaysFALSE" AND ("MODE SELECTION DB"."MODE BUFF" = 1);
END_REGION

REGION Network 95: PBV-123 VESSEL TOP DISH
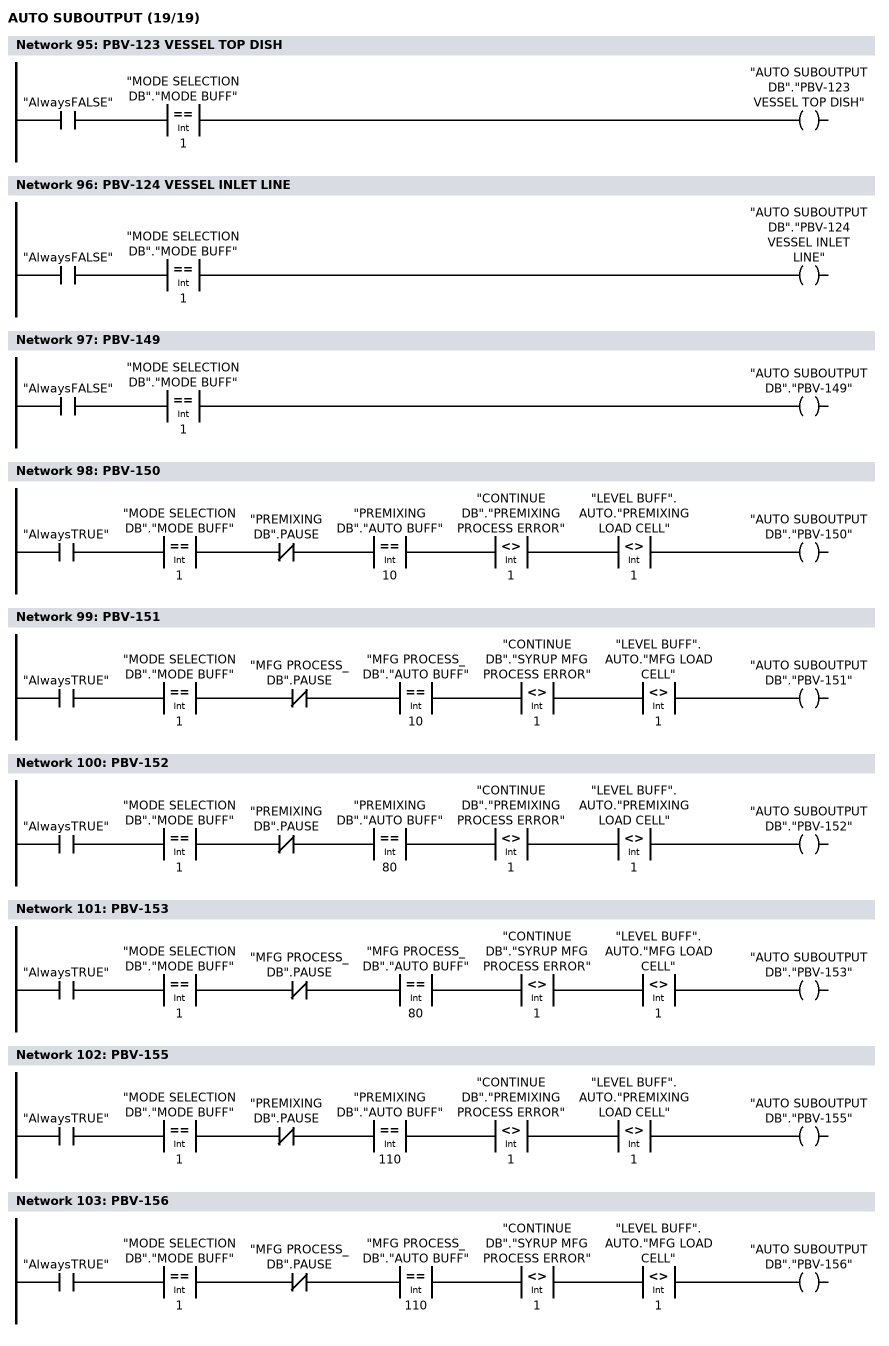
   RUNG wire#powerrail
      Contact( "AlwaysFALSE" )
      { S7_Templates := "SrcType := Int" } EQ_Contact(in1 := "MODE SELECTION DB"."MODE BUFF", in2 := 1)
      Coil( "AUTO SUBOUTPUT DB"."PBV-123 VESSEL TOP DISH" )
   END_RUNG
   // the same network as SCL:
   "AUTO SUBOUTPUT DB"."PBV-123 VESSEL TOP DISH" := "AlwaysFALSE" AND ("MODE SELECTION DB"."MODE BUFF" = 1);
END_REGION

REGION Network 96: PBV-124 VESSEL INLET LINE
   RUNG wire#powerrail
      Contact( "AlwaysFALSE" )
      { S7_Templates := "SrcType := Int" } EQ_Contact(in1 := "MODE SELECTION DB"."MODE BUFF", in2 := 1)
      Coil( "AUTO SUBOUTPUT DB"."PBV-124 VESSEL INLET LINE" )
   END_RUNG
   // the same network as SCL:
   "AUTO SUBOUTPUT DB"."PBV-124 VESSEL INLET LINE" := "AlwaysFALSE" AND ("MODE SELECTION DB"."MODE BUFF" = 1);
END_REGION

REGION Network 97: PBV-149
   RUNG wire#powerrail
      Contact( "AlwaysFALSE" )
      { S7_Templates := "SrcType := Int" } EQ_Contact(in1 := "MODE SELECTION DB"."MODE BUFF", in2 := 1)
      Coil( "AUTO SUBOUTPUT DB"."PBV-149" )
   END_RUNG
   // the same network as SCL:
   "AUTO SUBOUTPUT DB"."PBV-149" := "AlwaysFALSE" AND ("MODE SELECTION DB"."MODE BUFF" = 1);
END_REGION

REGION Network 98: PBV-150
   RUNG wire#powerrail
      Contact( "AlwaysTRUE" )
      { S7_Templates := "SrcType := Int" } EQ_Contact(in1 := "MODE SELECTION DB"."MODE BUFF", in2 := 1)
      I_Contact( "PREMIXING DB".PAUSE )
      { S7_Templates := "SrcType := Int" } EQ_Contact(in1 := "PREMIXING DB"."AUTO BUFF", in2 := 10)
      { S7_Templates := "SrcType := Int" } NE_Contact(in1 := "CONTINUE DB"."PREMIXING PROCESS ERROR", in2 := 1)
      { S7_Templates := "SrcType := Int" } NE_Contact(in1 := "LEVEL BUFF".AUTO."PREMIXING LOAD CELL", in2 := 1)
      Coil( "AUTO SUBOUTPUT DB"."PBV-150" )
   END_RUNG
   // the same network as SCL:
   "AUTO SUBOUTPUT DB"."PBV-150" := "AlwaysTRUE" AND ("MODE SELECTION DB"."MODE BUFF" = 1) AND NOT "PREMIXING DB".PAUSE AND ("PREMIXING DB"."AUTO BUFF" = 10) AND ("CONTINUE DB"."PREMIXING PROCESS ERROR" <> 1) AND ("LEVEL BUFF".AUTO."PREMIXING LOAD CELL" <> 1);
END_REGION

REGION Network 99: PBV-151
   RUNG wire#powerrail
      Contact( "AlwaysTRUE" )
      { S7_Templates := "SrcType := Int" } EQ_Contact(in1 := "MODE SELECTION DB"."MODE BUFF", in2 := 1)
      I_Contact( "MFG PROCESS_DB".PAUSE )
      { S7_Templates := "SrcType := Int" } EQ_Contact(in1 := "MFG PROCESS_DB"."AUTO BUFF", in2 := 10)
      { S7_Templates := "SrcType := Int" } NE_Contact(in1 := "CONTINUE DB"."SYRUP MFG PROCESS ERROR", in2 := 1)
      { S7_Templates := "SrcType := Int" } NE_Contact(in1 := "LEVEL BUFF".AUTO."MFG LOAD CELL", in2 := 1)
      Coil( "AUTO SUBOUTPUT DB"."PBV-151" )
   END_RUNG
   // the same network as SCL:
   "AUTO SUBOUTPUT DB"."PBV-151" := "AlwaysTRUE" AND ("MODE SELECTION DB"."MODE BUFF" = 1) AND NOT "MFG PROCESS_DB".PAUSE AND ("MFG PROCESS_DB"."AUTO BUFF" = 10) AND ("CONTINUE DB"."SYRUP MFG PROCESS ERROR" <> 1) AND ("LEVEL BUFF".AUTO."MFG LOAD CELL" <> 1);
END_REGION

REGION Network 100: PBV-152
   RUNG wire#powerrail
      Contact( "AlwaysTRUE" )
      { S7_Templates := "SrcType := Int" } EQ_Contact(in1 := "MODE SELECTION DB"."MODE BUFF", in2 := 1)
      I_Contact( "PREMIXING DB".PAUSE )
      { S7_Templates := "SrcType := Int" } EQ_Contact(in1 := "PREMIXING DB"."AUTO BUFF", in2 := 80)
      { S7_Templates := "SrcType := Int" } NE_Contact(in1 := "CONTINUE DB"."PREMIXING PROCESS ERROR", in2 := 1)
      { S7_Templates := "SrcType := Int" } NE_Contact(in1 := "LEVEL BUFF".AUTO."PREMIXING LOAD CELL", in2 := 1)
      Coil( "AUTO SUBOUTPUT DB"."PBV-152" )
   END_RUNG
   // the same network as SCL:
   "AUTO SUBOUTPUT DB"."PBV-152" := "AlwaysTRUE" AND ("MODE SELECTION DB"."MODE BUFF" = 1) AND NOT "PREMIXING DB".PAUSE AND ("PREMIXING DB"."AUTO BUFF" = 80) AND ("CONTINUE DB"."PREMIXING PROCESS ERROR" <> 1) AND ("LEVEL BUFF".AUTO."PREMIXING LOAD CELL" <> 1);
END_REGION

REGION Network 101: PBV-153
   RUNG wire#powerrail
      Contact( "AlwaysTRUE" )
      { S7_Templates := "SrcType := Int" } EQ_Contact(in1 := "MODE SELECTION DB"."MODE BUFF", in2 := 1)
      I_Contact( "MFG PROCESS_DB".PAUSE )
      { S7_Templates := "SrcType := Int" } EQ_Contact(in1 := "MFG PROCESS_DB"."AUTO BUFF", in2 := 80)
      { S7_Templates := "SrcType := Int" } NE_Contact(in1 := "CONTINUE DB"."SYRUP MFG PROCESS ERROR", in2 := 1)
      { S7_Templates := "SrcType := Int" } NE_Contact(in1 := "LEVEL BUFF".AUTO."MFG LOAD CELL", in2 := 1)
      Coil( "AUTO SUBOUTPUT DB"."PBV-153" )
   END_RUNG
   // the same network as SCL:
   "AUTO SUBOUTPUT DB"."PBV-153" := "AlwaysTRUE" AND ("MODE SELECTION DB"."MODE BUFF" = 1) AND NOT "MFG PROCESS_DB".PAUSE AND ("MFG PROCESS_DB"."AUTO BUFF" = 80) AND ("CONTINUE DB"."SYRUP MFG PROCESS ERROR" <> 1) AND ("LEVEL BUFF".AUTO."MFG LOAD CELL" <> 1);
END_REGION

REGION Network 102: PBV-155
   RUNG wire#powerrail
      Contact( "AlwaysTRUE" )
      { S7_Templates := "SrcType := Int" } EQ_Contact(in1 := "MODE SELECTION DB"."MODE BUFF", in2 := 1)
      I_Contact( "PREMIXING DB".PAUSE )
      { S7_Templates := "SrcType := Int" } EQ_Contact(in1 := "PREMIXING DB"."AUTO BUFF", in2 := 110)
      { S7_Templates := "SrcType := Int" } NE_Contact(in1 := "CONTINUE DB"."PREMIXING PROCESS ERROR", in2 := 1)
      { S7_Templates := "SrcType := Int" } NE_Contact(in1 := "LEVEL BUFF".AUTO."PREMIXING LOAD CELL", in2 := 1)
      Coil( "AUTO SUBOUTPUT DB"."PBV-155" )
   END_RUNG
   // the same network as SCL:
   "AUTO SUBOUTPUT DB"."PBV-155" := "AlwaysTRUE" AND ("MODE SELECTION DB"."MODE BUFF" = 1) AND NOT "PREMIXING DB".PAUSE AND ("PREMIXING DB"."AUTO BUFF" = 110) AND ("CONTINUE DB"."PREMIXING PROCESS ERROR" <> 1) AND ("LEVEL BUFF".AUTO."PREMIXING LOAD CELL" <> 1);
END_REGION

REGION Network 103: PBV-156
   RUNG wire#powerrail
      Contact( "AlwaysTRUE" )
      { S7_Templates := "SrcType := Int" } EQ_Contact(in1 := "MODE SELECTION DB"."MODE BUFF", in2 := 1)
      I_Contact( "MFG PROCESS_DB".PAUSE )
      { S7_Templates := "SrcType := Int" } EQ_Contact(in1 := "MFG PROCESS_DB"."AUTO BUFF", in2 := 110)
      { S7_Templates := "SrcType := Int" } NE_Contact(in1 := "CONTINUE DB"."SYRUP MFG PROCESS ERROR", in2 := 1)
      { S7_Templates := "SrcType := Int" } NE_Contact(in1 := "LEVEL BUFF".AUTO."MFG LOAD CELL", in2 := 1)
      Coil( "AUTO SUBOUTPUT DB"."PBV-156" )
   END_RUNG
   // the same network as SCL:
   "AUTO SUBOUTPUT DB"."PBV-156" := "AlwaysTRUE" AND ("MODE SELECTION DB"."MODE BUFF" = 1) AND NOT "MFG PROCESS_DB".PAUSE AND ("MFG PROCESS_DB"."AUTO BUFF" = 110) AND ("CONTINUE DB"."SYRUP MFG PROCESS ERROR" <> 1) AND ("LEVEL BUFF".AUTO."MFG LOAD CELL" <> 1);
END_REGION
END_FUNCTION
